LIN {X 0,Y 148.695,Z 336.424,A -85,B 0,C 180,E1 -24524.199,E2 -24524.199} C_VEL
LIN {X 0,Y 149.937,Z 338.136,A -85,B 0,C 180,E1 -24524.799,E2 -24524.799} C_VEL
LIN {X 0,Y 154.81,Z 345.559,A -85,B 0,C 180,E1 -24527.052,E2 -24527.052} C_VEL
LIN {X 0,Y 158.039,Z 351.12,A -85,B 0,C 180,E1 -24528.465,E2 -24528.465} C_VEL
LIN {X 0,Y 163.343,Z 362.974,A -85,B 0,C 180,E1 -24530.756,E2 -24530.756} C_VEL
LIN {X 0,Y 166.745,Z 372.421,A -85,B 0,C 180,E1 -24532.212,E2 -24532.212} C_VEL
LIN {X 0,Y 166.413,Z 382.188,A -85,B 0,C 180,E1 -24532.644,E2 -24532.644} C_VEL
LIN {X 0,Y 165.211,Z 401.171,A -85,B 0,C 180,E1 -24533.449,E2 -24533.449} C_VEL
LIN {X 0,Y 163.851,Z 412.228,A -85,B 0,C 180,E1 -24534.244,E2 -24534.244} C_VEL
LIN {X 0,Y 161.723,Z 423.778,A -85,B 0,C 180,E1 -24535.603,E2 -24535.603} C_VEL
LIN {X 0,Y 159.816,Z 431.992,A -85,B 0,C 180,E1 -24536.921,E2 -24536.921} C_VEL
LIN {X 0,Y 157.688,Z 439.473,A -85,B 0,C 180,E1 -24538.421,E2 -24538.421} C_VEL
LIN {X 0,Y 155.05,Z 447.512,A -85,B 0,C 180,E1 -24540.467,E2 -24540.467} C_VEL
LIN {X 0,Y 152.63,Z 454.152,A -85,B 0,C 180,E1 -24542.584,E2 -24542.584} C_VEL
LIN {X 0,Y 150.051,Z 460.455,A -85,B 0,C 180,E1 -24545.069,E2 -24545.069} C_VEL
LIN {X 0,Y 147.775,Z 465.69,A -85,B 0,C 180,E1 -24547.638,E2 -24547.638} C_VEL
LIN {X 0,Y 145.868,Z 470.055,A -85,B 0,C 180,E1 -24550.29,E2 -24550.29} C_VEL
LIN {X 0,Y 143.545,Z 475.202,A -85,B 0,C 180,E1 -24554.379,E2 -24554.379} C_VEL
LIN {X 0,Y 141.917,Z 478.977,A -85,B 0,C 180,E1 -24558.575,E2 -24558.575} C_VEL
LIN {X 0,Y 141.219,Z 480.707,A -85,B 0,C 180,E1 -24561.414,E2 -24561.414} C_VEL
LIN {X 0,Y 140.732,Z 481.944,A -85,B 0,C 180,E1 -24564.268,E2 -24564.268} C_VEL
LIN {X 0,Y 140.537,Z 482.711,A -85,B 0,C 180,E1 -24567.134,E2 -24567.134} C_VEL
LIN {X 0,Y 140.501,Z 483,A -85,B 0,C 180,E1 -24570,E2 -24570} C_VEL
LIN {X 0,Y 140.537,Z 482.7,A -85,B 0,C 180,E1 -24572.866,E2 -24572.866} C_VEL
LIN {X 0,Y 140.727,Z 481.911,A -85,B 0,C 180,E1 -24575.732,E2 -24575.732} C_VEL
LIN {X 0,Y 141.165,Z 480.651,A -85,B 0,C 180,E1 -24578.589,E2 -24578.589} C_VEL
LIN {X 0,Y 142.391,Z 477.747,A -85,B 0,C 180,E1 -24582.832,E2 -24582.832} C_VEL
LIN {X 0,Y 143.538,Z 475.097,A -85,B 0,C 180,E1 -24585.622,E2 -24585.622} C_VEL
LIN {X 0,Y 145.852,Z 469.92,A -85,B 0,C 180,E1 -24589.712,E2 -24589.712} C_VEL
LIN {X 0,Y 147.47,Z 466.222,A -85,B 0,C 180,E1 -24591.972,E2 -24591.972} C_VEL
LIN {X 0,Y 148.291,Z 462.951,A -85,B 0,C 180,E1 -24593.828,E2 -24593.828} C_VEL
LIN {X 0,Y 148.181,Z 457.047,A -85,B 0,C 180,E1 -24596.903,E2 -24596.903} C_VEL
LIN {X 0,Y 148.279,Z 450.489,A -85,B 0,C 180,E1 -24599.774,E2 -24599.774} C_VEL
LIN {X 0,Y 149.393,Z 445.99,A -85,B 0,C 180,E1 -24601.248,E2 -24601.248} C_VEL
LIN {X 0,Y 152.515,Z 436.512,A -85,B 0,C 180,E1 -24603.57,E2 -24603.57} C_VEL
LIN {X 0,Y 154.97,Z 427.195,A -85,B 0,C 180,E1 -24605.283,E2 -24605.283} C_VEL
LIN {X 0,Y 157.011,Z 417.741,A -85,B 0,C 180,E1 -24606.577,E2 -24606.577} C_VEL
LIN {X 0,Y 158.536,Z 408.45,A -85,B 0,C 180,E1 -24607.495,E2 -24607.495} C_VEL
LIN {X 0,Y 159.576,Z 399.713,A -85,B 0,C 180,E1 -24608.066,E2 -24608.066} C_VEL
LIN {X 0,Y 161.057,Z 374.2,A -85,B 0,C 180,E1 -24609.16,E2 -24609.16} C_VEL
LIN {X 0,Y 156.299,Z 361.781,A -85,B 0,C 180,E1 -24611.334,E2 -24611.334} C_VEL
LIN {X 0,Y 152.216,Z 352.913,A -85,B 0,C 180,E1 -24613.26,E2 -24613.26} C_VEL
LIN {X 0,Y 145.462,Z 342.285,A -85,B 0,C 180,E1 -24616.558,E2 -24616.558} C_VEL
LIN {X 0,Y 142.86,Z 338.543,A -85,B 0,C 180,E1 -24617.945,E2 -24617.945} C_VEL
LIN {X 0,Y 140.098,Z 334.863,A -85,B 0,C 180,E1 -24619.495,E2 -24619.495} C_VEL
LIN {X 0,Y 139.28,Z 333.439,A -85,B 0,C 180,E1 -24620.002,E2 -24620.002} C_VEL
LIN {X 0,Y 137.047,Z 331.169,A -85,B 0,C 180,E1 -24621.313,E2 -24621.313} C_VEL
LIN {X 0,Y 136.131,Z 328.935,A -85,B 0,C 180,E1 -24622.189,E2 -24622.189} C_VEL
LIN {X 0,Y 136.019,Z 328.352,A -85,B 0,C 180,E1 -24623.083,E2 -24623.083} C_VEL
LIN {X 0,Y 136.079,Z 328.326,A -85,B 0,C 180,E1 -24625.723,E2 -24625.723} C_VEL
LIN {X 0,Y 136.114,Z 328.328,A -85,B 0,C 180,E1 -24632.31,E2 -24632.31} C_VEL
LIN {X 0,Y 136.18,Z 328.306,A -85,B 0,C 180,E1 -24638.823,E2 -24638.823} C_VEL
LIN {X 0,Y 136.218,Z 328.297,A -85,B 0,C 180,E1 -24645.051,E2 -24645.051} C_VEL
LIN {X 0,Y 136.422,Z 328.278,A -85,B 0,C 180,E1 -24648.179,E2 -24648.179} C_VEL
LIN {X 0,Y 136.541,Z 328.288,A -85,B 0,C 180,E1 -24651.117,E2 -24651.117} C_VEL
LIN {X 0,Y 137.105,Z 328.22,A -85,B 0,C 180,E1 -24660,E2 -24660} C_VEL
LIN {X 0,Y 136.529,Z 328.289,A -85,B 0,C 180,E1 -24668.884,E2 -24668.884} C_VEL
LIN {X 0,Y 136.41,Z 328.279,A -85,B 0,C 180,E1 -24671.893,E2 -24671.893} C_VEL
LIN {X 0,Y 136.162,Z 328.337,A -85,B 0,C 180,E1 -24678.041,E2 -24678.041} C_VEL
LIN {X 0,Y 136.143,Z 328.308,A -85,B 0,C 180,E1 -24681.693,E2 -24681.693} C_VEL
LIN {X 0,Y 136.085,Z 328.324,A -85,B 0,C 180,E1 -24688.606,E2 -24688.606} C_VEL
LIN {X 0,Y 136.066,Z 328.321,A -85,B 0,C 180,E1 -24694.623,E2 -24694.623} C_VEL
LIN {X 0,Y 136.059,Z 328.636,A -85,B 0,C 180,E1 -24697.544,E2 -24697.544} C_VEL
LIN {X 0,Y 136.414,Z 329.867,A -85,B 0,C 180,E1 -24698.264,E2 -24698.264} C_VEL
LIN {X 0,Y 138.033,Z 332.419,A -85,B 0,C 180,E1 -24699.341,E2 -24699.341} C_VEL
LIN {X 0,Y 139.651,Z 333.976,A -85,B 0,C 180,E1 -24700.266,E2 -24700.266} C_VEL
LIN {X 0,Y 141.692,Z 337.197,A -85,B 0,C 180,E1 -24701.474,E2 -24701.474} C_VEL
LIN {X 0,Y 142.993,Z 338.765,A -85,B 0,C 180,E1 -24702.175,E2 -24702.175} C_VEL
LIN {X 0,Y 148.809,Z 347.525,A -85,B 0,C 180,E1 -24705.181,E2 -24705.181} C_VEL
LIN {X 0,Y 153.169,Z 354.766,A -85,B 0,C 180,E1 -24707.235,E2 -24707.235} C_VEL
LIN {X 0,Y 157.306,Z 364.284,A -85,B 0,C 180,E1 -24709.18,E2 -24709.18} C_VEL
LIN {X 0,Y 161.073,Z 374.306,A -85,B 0,C 180,E1 -24710.895,E2 -24710.895} C_VEL
LIN {X 0,Y 159.461,Z 400.566,A -85,B 0,C 180,E1 -24712.012,E2 -24712.012} C_VEL
LIN {X 0,Y 158.152,Z 411.086,A -85,B 0,C 180,E1 -24712.761,E2 -24712.761} C_VEL
LIN {X 0,Y 155.974,Z 423.044,A -85,B 0,C 180,E1 -24714.144,E2 -24714.144} C_VEL
LIN {X 0,Y 153.613,Z 432.702,A -85,B 0,C 180,E1 -24715.745,E2 -24715.745} C_VEL
LIN {X 0,Y 151.353,Z 440.221,A -85,B 0,C 180,E1 -24717.331,E2 -24717.331} C_VEL
LIN {X 0,Y 148.95,Z 447.117,A -85,B 0,C 180,E1 -24719.129,E2 -24719.129} C_VEL
LIN {X 0,Y 146.422,Z 453.821,A -85,B 0,C 180,E1 -24721.317,E2 -24721.317} C_VEL
LIN {X 0,Y 143.695,Z 460.173,A -85,B 0,C 180,E1 -24723.885,E2 -24723.885} C_VEL
LIN {X 0,Y 141.259,Z 465.454,A -85,B 0,C 180,E1 -24726.546,E2 -24726.546} C_VEL
LIN {X 0,Y 139.225,Z 469.863,A -85,B 0,C 180,E1 -24729.308,E2 -24729.308} C_VEL
LIN {X 0,Y 136.733,Z 475.052,A -85,B 0,C 180,E1 -24733.579,E2 -24733.579} C_VEL
LIN {X 0,Y 135.505,Z 477.712,A -85,B 0,C 180,E1 -24736.503,E2 -24736.503} C_VEL
LIN {X 0,Y 134.143,Z 480.627,A -85,B 0,C 180,E1 -24740.957,E2 -24740.957} C_VEL
LIN {X 0,Y 133.662,Z 481.896,A -85,B 0,C 180,E1 -24743.964,E2 -24743.964} C_VEL
LIN {X 0,Y 133.466,Z 482.695,A -85,B 0,C 180,E1 -24746.982,E2 -24746.982} C_VEL
LIN {X 0,Y 133.419,Z 482.999,A -85,B 0,C 180,E1 -24750,E2 -24750} C_VEL
LIN {X 0,Y 133.466,Z 482.716,A -85,B 0,C 180,E1 -24753.018,E2 -24753.018} C_VEL
LIN {X 0,Y 133.662,Z 481.959,A -85,B 0,C 180,E1 -24756.036,E2 -24756.036} C_VEL
LIN {X 0,Y 134.142,Z 480.732,A -85,B 0,C 180,E1 -24759.043,E2 -24759.043} C_VEL
LIN {X 0,Y 135.48,Z 477.861,A -85,B 0,C 180,E1 -24763.499,E2 -24763.499} C_VEL
LIN {X 0,Y 136.68,Z 475.247,A -85,B 0,C 180,E1 -24766.427,E2 -24766.427} C_VEL
LIN {X 0,Y 139.185,Z 470.112,A -85,B 0,C 180,E1 -24770.698,E2 -24770.698} C_VEL
LIN {X 0,Y 141.795,Z 464.588,A -85,B 0,C 180,E1 -24774.136,E2 -24774.136} C_VEL
LIN {X 0,Y 144.923,Z 457.644,A -85,B 0,C 180,E1 -24777.432,E2 -24777.432} C_VEL
LIN {X 0,Y 148.155,Z 449.673,A -85,B 0,C 180,E1 -24780.265,E2 -24780.265} C_VEL
LIN {X 0,Y 150.871,Z 442.075,A -85,B 0,C 180,E1 -24782.391,E2 -24782.391} C_VEL
LIN {X 0,Y 153.042,Z 435.345,A -85,B 0,C 180,E1 -24783.903,E2 -24783.903} C_VEL
LIN {X 0,Y 155.42,Z 426.284,A -85,B 0,C 180,E1 -24785.516,E2 -24785.516} C_VEL
LIN {X 0,Y 157.213,Z 417.303,A -85,B 0,C 180,E1 -24786.753,E2 -24786.753} C_VEL
LIN {X 0,Y 158.785,Z 407.979,A -85,B 0,C 180,E1 -24787.641,E2 -24787.641} C_VEL
LIN {X 0,Y 159.771,Z 398.211,A -85,B 0,C 180,E1 -24788.286,E2 -24788.286} C_VEL
LIN {X 0,Y 161.177,Z 374.379,A -85,B 0,C 180,E1 -24789.275,E2 -24789.275} C_VEL
LIN {X 0,Y 156.324,Z 361.554,A -85,B 0,C 180,E1 -24791.51,E2 -24791.51} C_VEL
LIN {X 0,Y 152.125,Z 352.746,A -85,B 0,C 180,E1 -24793.483,E2 -24793.483} C_VEL
LIN {X 0,Y 145.533,Z 342.329,A -85,B 0,C 180,E1 -24796.725,E2 -24796.725} C_VEL
LIN {X 0,Y 142.997,Z 338.745,A -85,B 0,C 180,E1 -24798.077,E2 -24798.077} C_VEL
LIN {X 0,Y 140.121,Z 334.906,A -85,B 0,C 180,E1 -24799.7,E2 -24799.7} C_VEL
LIN {X 0,Y 139.31,Z 333.464,A -85,B 0,C 180,E1 -24800.208,E2 -24800.208} C_VEL
LIN {X 0,Y 137.107,Z 331.257,A -85,B 0,C 180,E1 -24801.507,E2 -24801.507} C_VEL
LIN {X 0,Y 136.142,Z 328.931,A -85,B 0,C 180,E1 -24802.425,E2 -24802.425} C_VEL
LIN {X 0,Y 136.037,Z 328.331,A -85,B 0,C 180,E1 -24803.55,E2 -24803.55} C_VEL
LIN {X 0,Y 136.051,Z 328.33,A -85,B 0,C 180,E1 -24808.897,E2 -24808.897} C_VEL
LIN {X 0,Y 136.115,Z 328.326,A -85,B 0,C 180,E1 -24812.309,E2 -24812.309} C_VEL
LIN {X 0,Y 136.181,Z 328.305,A -85,B 0,C 180,E1 -24818.822,E2 -24818.822} C_VEL
LIN {X 0,Y 136.218,Z 328.298,A -85,B 0,C 180,E1 -24825.05,E2 -24825.05} C_VEL
LIN {X 0,Y 136.423,Z 328.277,A -85,B 0,C 180,E1 -24828.178,E2 -24828.178} C_VEL
LIN {X 0,Y 136.541,Z 328.288,A -85,B 0,C 180,E1 -24831.117,E2 -24831.117} C_VEL
LIN {X 0,Y 137.105,Z 328.22,A -85,B 0,C 180,E1 -24840,E2 -24840} C_VEL
LIN {X 0,Y 136.529,Z 328.289,A -85,B 0,C 180,E1 -24848.883,E2 -24848.883} C_VEL
LIN {X 0,Y 136.41,Z 328.278,A -85,B 0,C 180,E1 -24851.893,E2 -24851.893} C_VEL
LIN {X 0,Y 136.161,Z 328.337,A -85,B 0,C 180,E1 -24858.04,E2 -24858.04} C_VEL
LIN {X 0,Y 136.143,Z 328.308,A -85,B 0,C 180,E1 -24861.693,E2 -24861.693} C_VEL
LIN {X 0,Y 136.084,Z 328.323,A -85,B 0,C 180,E1 -24868.605,E2 -24868.605} C_VEL
LIN {X 0,Y 136.043,Z 328.32,A -85,B 0,C 180,E1 -24874.629,E2 -24874.629} C_VEL
LIN {X 0,Y 136.057,Z 328.64,A -85,B 0,C 180,E1 -24877.31,E2 -24877.31} C_VEL
LIN {X 0,Y 136.449,Z 329.96,A -85,B 0,C 180,E1 -24878.058,E2 -24878.058} C_VEL
LIN {X 0,Y 138.064,Z 332.476,A -85,B 0,C 180,E1 -24879.133,E2 -24879.133} C_VEL
LIN {X 0,Y 139.681,Z 333.957,A -85,B 0,C 180,E1 -24880.058,E2 -24880.058} C_VEL
LIN {X 0,Y 141.743,Z 337.249,A -85,B 0,C 180,E1 -24881.288,E2 -24881.288} C_VEL
LIN {X 0,Y 143.034,Z 338.862,A -85,B 0,C 180,E1 -24881.993,E2 -24881.993} C_VEL
LIN {X 0,Y 148.483,Z 346.884,A -85,B 0,C 180,E1 -24884.822,E2 -24884.822} C_VEL
LIN {X 0,Y 153.376,Z 355.105,A -85,B 0,C 180,E1 -24887.151,E2 -24887.151} C_VEL
LIN {X 0,Y 158.553,Z 367.079,A -85,B 0,C 180,E1 -24889.566,E2 -24889.566} C_VEL
LIN {X 0,Y 161.175,Z 374.479,A -85,B 0,C 180,E1 -24890.775,E2 -24890.775} C_VEL
LIN {X 0,Y 159.576,Z 401.187,A -85,B 0,C 180,E1 -24891.934,E2 -24891.934} C_VEL
LIN {X 0,Y 158.064,Z 412.877,A -85,B 0,C 180,E1 -24892.806,E2 -24892.806} C_VEL
LIN {X 0,Y 155.92,Z 423.784,A -85,B 0,C 180,E1 -24894.13,E2 -24894.13} C_VEL
LIN {X 0,Y 153.706,Z 432.765,A -85,B 0,C 180,E1 -24895.628,E2 -24895.628} C_VEL
LIN {X 0,Y 151.277,Z 440.706,A -85,B 0,C 180,E1 -24897.312,E2 -24897.312} C_VEL
LIN {X 0,Y 148.545,Z 448.536,A -85,B 0,C 180,E1 -24899.43,E2 -24899.43} C_VEL
LIN {X 0,Y 145.646,Z 455.858,A -85,B 0,C 180,E1 -24901.936,E2 -24901.936} C_VEL
LIN {X 0,Y 142.4,Z 463.284,A -85,B 0,C 180,E1 -24905.197,E2 -24905.197} C_VEL
LIN {X 0,Y 139.71,Z 469.1,A -85,B 0,C 180,E1 -24908.611,E2 -24908.611} C_VEL
LIN {X 0,Y 137.458,Z 473.686,A -85,B 0,C 180,E1 -24912.136,E2 -24912.136} C_VEL
LIN {X 0,Y 136.064,Z 476.666,A -85,B 0,C 180,E1 -24915.034,E2 -24915.034} C_VEL
LIN {X 0,Y 134.962,Z 478.978,A -85,B 0,C 180,E1 -24917.978,E2 -24917.978} C_VEL
LIN {X 0,Y 134.184,Z 480.708,A -85,B 0,C 180,E1 -24920.96,E2 -24920.96} C_VEL
LIN {X 0,Y 133.667,Z 481.945,A -85,B 0,C 180,E1 -24923.964,E2 -24923.964} C_VEL
LIN {X 0,Y 133.464,Z 482.711,A -85,B 0,C 180,E1 -24926.982,E2 -24926.982} C_VEL
LIN {X 0,Y 133.418,Z 483,A -85,B 0,C 180,E1 -24930,E2 -24930} C_VEL
LIN {X 0,Y 133.464,Z 482.7,A -85,B 0,C 180,E1 -24933.018,E2 -24933.018} C_VEL
LIN {X 0,Y 133.661,Z 481.911,A -85,B 0,C 180,E1 -24936.036,E2 -24936.036} C_VEL
LIN {X 0,Y 134.141,Z 480.651,A -85,B 0,C 180,E1 -24939.043,E2 -24939.043} C_VEL
LIN {X 0,Y 135.482,Z 477.746,A -85,B 0,C 180,E1 -24943.499,E2 -24943.499} C_VEL
LIN {X 0,Y 136.7,Z 475.096,A -85,B 0,C 180,E1 -24946.425,E2 -24946.425} C_VEL
LIN {X 0,Y 139.176,Z 469.919,A -85,B 0,C 180,E1 -24950.7,E2 -24950.7} C_VEL
LIN {X 0,Y 142.4,Z 463.086,A -85,B 0,C 180,E1 -24954.803,E2 -24954.803} C_VEL
LIN {X 0,Y 145.648,Z 455.62,A -85,B 0,C 180,E1 -24958.064,E2 -24958.064} C_VEL
LIN {X 0,Y 148.533,Z 448.254,A -85,B 0,C 180,E1 -24960.573,E2 -24960.573} C_VEL
LIN {X 0,Y 149.393,Z 445.99,A -85,B 0,C 180,E1 -24961.248,E2 -24961.248} C_VEL
LIN {X 0,Y 150.48,Z 441.43,A -85,B 0,C 180,E1 -24962.633,E2 -24962.633} C_VEL
LIN {X 0,Y 150.534,Z 433.661,A -85,B 0,C 180,E1 -24964.998,E2 -24964.998} C_VEL
LIN {X 0,Y 150.331,Z 425.341,A -85,B 0,C 180,E1 -24967.057,E2 -24967.057} C_VEL
LIN {X 0,Y 150.947,Z 419.921,A -85,B 0,C 180,E1 -24967.922,E2 -24967.922} C_VEL
LIN {X 0,Y 152.843,Z 409.396,A -85,B 0,C 180,E1 -24969.029,E2 -24969.029} C_VEL
LIN {X 0,Y 154.058,Z 399.697,A -85,B 0,C 180,E1 -24969.691,E2 -24969.691} C_VEL
LIN {X 0,Y 155.493,Z 376.136,A -85,B 0,C 180,E1 -24970.733,E2 -24970.733} C_VEL
LIN {X 0,Y 151.514,Z 365.491,A -85,B 0,C 180,E1 -24972.71,E2 -24972.71} C_VEL
LIN {X 0,Y 147.907,Z 357.529,A -85,B 0,C 180,E1 -24974.542,E2 -24974.542} C_VEL
LIN {X 0,Y 141.823,Z 347.659,A -85,B 0,C 180,E1 -24977.734,E2 -24977.734} C_VEL
LIN {X 0,Y 138.092,Z 342.464,A -85,B 0,C 180,E1 -24979.874,E2 -24979.874} C_VEL
LIN {X 0,Y 135.728,Z 338.996,A -85,B 0,C 180,E1 -24981.359,E2 -24981.359} C_VEL
LIN {X 0,Y 133.34,Z 335.935,A -85,B 0,C 180,E1 -24982.927,E2 -24982.927} C_VEL
LIN {X 0,Y 132.436,Z 334.429,A -85,B 0,C 180,E1 -24983.581,E2 -24983.581} C_VEL
LIN {X 0,Y 130.24,Z 332.395,A -85,B 0,C 180,E1 -24985.103,E2 -24985.103} C_VEL
LIN {X 0,Y 129.116,Z 329.851,A -85,B 0,C 180,E1 -24986.308,E2 -24986.308} C_VEL
LIN {X 0,Y 128.997,Z 329.255,A -85,B 0,C 180,E1 -24987.452,E2 -24987.452} C_VEL
LIN {X 0,Y 129.014,Z 329.201,A -85,B 0,C 180,E1 -24990.642,E2 -24990.642} C_VEL
LIN {X 0,Y 128.995,Z 329.229,A -85,B 0,C 180,E1 -24994.16,E2 -24994.16} C_VEL
LIN {X 0,Y 129.065,Z 329.188,A -85,B 0,C 180,E1 -24997.771,E2 -24997.771} C_VEL
LIN {X 0,Y 129.141,Z 329.184,A -85,B 0,C 180,E1 -25004.211,E2 -25004.211} C_VEL
LIN {X 0,Y 129.34,Z 329.156,A -85,B 0,C 180,E1 -25007.974,E2 -25007.974} C_VEL
LIN {X 0,Y 129.465,Z 329.17,A -85,B 0,C 180,E1 -25010.628,E2 -25010.628} C_VEL
LIN {X 0,Y 130.06,Z 329.098,A -85,B 0,C 180,E1 -25020,E2 -25020} C_VEL
LIN {X 0,Y 129.456,Z 329.171,A -85,B 0,C 180,E1 -25029.374,E2 -25029.374} C_VEL
LIN {X 0,Y 129.294,Z 329.158,A -85,B 0,C 180,E1 -25032.558,E2 -25032.558} C_VEL
LIN {X 0,Y 129.079,Z 329.211,A -85,B 0,C 180,E1 -25039.068,E2 -25039.068} C_VEL
LIN {X 0,Y 129.039,Z 329.192,A -85,B 0,C 180,E1 -25042.411,E2 -25042.411} C_VEL
LIN {X 0,Y 128.995,Z 329.228,A -85,B 0,C 180,E1 -25045.84,E2 -25045.84} C_VEL
LIN {X 0,Y 129.001,Z 329.207,A -85,B 0,C 180,E1 -25051.169,E2 -25051.169} C_VEL
LIN {X 0,Y 129.048,Z 329.596,A -85,B 0,C 180,E1 -25053.474,E2 -25053.474} C_VEL
LIN {X 0,Y 129.49,Z 330.922,A -85,B 0,C 180,E1 -25054.3,E2 -25054.3} C_VEL
LIN {X 0,Y 131.021,Z 333.346,A -85,B 0,C 180,E1 -25055.516,E2 -25055.516} C_VEL
LIN {X 0,Y 132.865,Z 334.901,A -85,B 0,C 180,E1 -25056.755,E2 -25056.755} C_VEL
LIN {X 0,Y 134.824,Z 338.072,A -85,B 0,C 180,E1 -25058.126,E2 -25058.126} C_VEL
LIN {X 0,Y 136.468,Z 339.947,A -85,B 0,C 180,E1 -25059.151,E2 -25059.151} C_VEL
LIN {X 0,Y 138.92,Z 343.431,A -85,B 0,C 180,E1 -25060.649,E2 -25060.649} C_VEL
LIN {X 0,Y 144.623,Z 352.07,A -85,B 0,C 180,E1 -25063.827,E2 -25063.827} C_VEL
LIN {X 0,Y 148.928,Z 359.491,A -85,B 0,C 180,E1 -25066.017,E2 -25066.017} C_VEL
LIN {X 0,Y 153.362,Z 370.157,A -85,B 0,C 180,E1 -25068.256,E2 -25068.256} C_VEL
LIN {X 0,Y 155.505,Z 376.196,A -85,B 0,C 180,E1 -25069.319,E2 -25069.319} C_VEL
LIN {X 0,Y 153.894,Z 401.036,A -85,B 0,C 180,E1 -25070.413,E2 -25070.413} C_VEL
LIN {X 0,Y 152.457,Z 411.896,A -85,B 0,C 180,E1 -25071.218,E2 -25071.218} C_VEL
LIN {X 0,Y 150.279,Z 423.05,A -85,B 0,C 180,E1 -25072.559,E2 -25072.559} C_VEL
LIN {X 0,Y 147.966,Z 432.158,A -85,B 0,C 180,E1 -25074.089,E2 -25074.089} C_VEL
LIN {X 0,Y 145.441,Z 440.225,A -85,B 0,C 180,E1 -25075.825,E2 -25075.825} C_VEL
LIN {X 0,Y 142.892,Z 447.12,A -85,B 0,C 180,E1 -25077.665,E2 -25077.665} C_VEL
LIN {X 0,Y 140.247,Z 453.824,A -85,B 0,C 180,E1 -25079.927,E2 -25079.927} C_VEL
LIN {X 0,Y 137.352,Z 460.176,A -85,B 0,C 180,E1 -25082.581,E2 -25082.581} C_VEL
LIN {X 0,Y 134.779,Z 465.456,A -85,B 0,C 180,E1 -25085.345,E2 -25085.345} C_VEL
LIN {X 0,Y 132.592,Z 469.865,A -85,B 0,C 180,E1 -25088.221,E2 -25088.221} C_VEL
LIN {X 0,Y 129.931,Z 475.053,A -85,B 0,C 180,E1 -25092.693,E2 -25092.693} C_VEL
LIN {X 0,Y 128.595,Z 477.713,A -85,B 0,C 180,E1 -25095.763,E2 -25095.763} C_VEL
LIN {X 0,Y 127.143,Z 480.627,A -85,B 0,C 180,E1 -25100.455,E2 -25100.455} C_VEL
LIN {X 0,Y 126.595,Z 481.897,A -85,B 0,C 180,E1 -25103.625,E2 -25103.625} C_VEL
LIN {X 0,Y 126.382,Z 482.695,A -85,B 0,C 180,E1 -25106.812,E2 -25106.812} C_VEL
LIN {X 0,Y 126.322,Z 482.999,A -85,B 0,C 180,E1 -25110,E2 -25110} C_VEL
LIN {X 0,Y 126.382,Z 482.716,A -85,B 0,C 180,E1 -25113.188,E2 -25113.188} C_VEL
LIN {X 0,Y 126.595,Z 481.959,A -85,B 0,C 180,E1 -25116.375,E2 -25116.375} C_VEL
LIN {X 0,Y 127.142,Z 480.731,A -85,B 0,C 180,E1 -25119.545,E2 -25119.545} C_VEL
LIN {X 0,Y 128.57,Z 477.86,A -85,B 0,C 180,E1 -25124.24,E2 -25124.24} C_VEL
LIN {X 0,Y 129.883,Z 475.246,A -85,B 0,C 180,E1 -25127.314,E2 -25127.314} C_VEL
LIN {X 0,Y 132.555,Z 470.11,A -85,B 0,C 180,E1 -25131.785,E2 -25131.785} C_VEL
LIN {X 0,Y 135.33,Z 464.586,A -85,B 0,C 180,E1 -25135.368,E2 -25135.368} C_VEL
LIN {X 0,Y 138.659,Z 457.641,A -85,B 0,C 180,E1 -25138.783,E2 -25138.783} C_VEL
LIN {X 0,Y 142.064,Z 449.67,A -85,B 0,C 180,E1 -25141.709,E2 -25141.709} C_VEL
LIN {X 0,Y 144.94,Z 442.071,A -85,B 0,C 180,E1 -25143.891,E2 -25143.891} C_VEL
LIN {X 0,Y 147.528,Z 434.049,A -85,B 0,C 180,E1 -25145.716,E2 -25145.716} C_VEL
LIN {X 0,Y 149.854,Z 425.655,A -85,B 0,C 180,E1 -25147.19,E2 -25147.19} C_VEL
LIN {X 0,Y 151.7,Z 416.639,A -85,B 0,C 180,E1 -25148.439,E2 -25148.439} C_VEL
LIN {X 0,Y 153.358,Z 406.897,A -85,B 0,C 180,E1 -25149.359,E2 -25149.359} C_VEL
LIN {X 0,Y 154.572,Z 394.44,A -85,B 0,C 180,E1 -25150.102,E2 -25150.102} C_VEL
LIN {X 0,Y 155.669,Z 376.382,A -85,B 0,C 180,E1 -25150.832,E2 -25150.832} C_VEL
LIN {X 0,Y 151.079,Z 364.134,A -85,B 0,C 180,E1 -25153.129,E2 -25153.129} C_VEL
LIN {X 0,Y 147.817,Z 357.328,A -85,B 0,C 180,E1 -25154.779,E2 -25154.779} C_VEL
LIN {X 0,Y 141.871,Z 347.69,A -85,B 0,C 180,E1 -25157.92,E2 -25157.92} C_VEL
LIN {X 0,Y 138.318,Z 342.743,A -85,B 0,C 180,E1 -25159.965,E2 -25159.965} C_VEL
LIN {X 0,Y 135.902,Z 339.167,A -85,B 0,C 180,E1 -25161.488,E2 -25161.488} C_VEL
LIN {X 0,Y 133.584,Z 336.285,A -85,B 0,C 180,E1 -25163.005,E2 -25163.005} C_VEL
LIN {X 0,Y 132.702,Z 334.585,A -85,B 0,C 180,E1 -25163.665,E2 -25163.665} C_VEL
LIN {X 0,Y 130.37,Z 332.591,A -85,B 0,C 180,E1 -25165.27,E2 -25165.27} C_VEL
LIN {X 0,Y 129.117,Z 329.902,A -85,B 0,C 180,E1 -25166.55,E2 -25166.55} C_VEL
LIN {X 0,Y 128.989,Z 329.282,A -85,B 0,C 180,E1 -25167.449,E2 -25167.449} C_VEL
LIN {X 0,Y 129.015,Z 329.2,A -85,B 0,C 180,E1 -25170.641,E2 -25170.641} C_VEL
LIN {X 0,Y 128.995,Z 329.23,A -85,B 0,C 180,E1 -25174.16,E2 -25174.16} C_VEL
LIN {X 0,Y 129.066,Z 329.188,A -85,B 0,C 180,E1 -25177.77,E2 -25177.77} C_VEL
LIN {X 0,Y 129.141,Z 329.185,A -85,B 0,C 180,E1 -25184.21,E2 -25184.21} C_VEL
LIN {X 0,Y 129.34,Z 329.156,A -85,B 0,C 180,E1 -25187.973,E2 -25187.973} C_VEL
LIN {X 0,Y 129.465,Z 329.17,A -85,B 0,C 180,E1 -25190.627,E2 -25190.627} C_VEL
LIN {X 0,Y 130.06,Z 329.098,A -85,B 0,C 180,E1 -25200,E2 -25200} C_VEL
LIN {X 0,Y 129.456,Z 329.171,A -85,B 0,C 180,E1 -25209.373,E2 -25209.373} C_VEL
LIN {X 0,Y 129.294,Z 329.158,A -85,B 0,C 180,E1 -25212.558,E2 -25212.558} C_VEL
LIN {X 0,Y 129.078,Z 329.21,A -85,B 0,C 180,E1 -25219.067,E2 -25219.067} C_VEL
LIN {X 0,Y 129.039,Z 329.192,A -85,B 0,C 180,E1 -25222.411,E2 -25222.411} C_VEL
LIN {X 0,Y 128.995,Z 329.229,A -85,B 0,C 180,E1 -25225.84,E2 -25225.84} C_VEL
LIN {X 0,Y 128.999,Z 329.208,A -85,B 0,C 180,E1 -25231.169,E2 -25231.169} C_VEL
LIN {X 0,Y 129.054,Z 329.632,A -85,B 0,C 180,E1 -25233.231,E2 -25233.231} C_VEL
LIN {X 0,Y 129.501,Z 331.019,A -85,B 0,C 180,E1 -25234.047,E2 -25234.047} C_VEL
LIN {X 0,Y 131.127,Z 333.468,A -85,B 0,C 180,E1 -25235.331,E2 -25235.331} C_VEL
LIN {X 0,Y 132.878,Z 334.934,A -85,B 0,C 180,E1 -25236.514,E2 -25236.514} C_VEL
LIN {X 0,Y 134.946,Z 338.233,A -85,B 0,C 180,E1 -25237.966,E2 -25237.966} C_VEL
LIN {X 0,Y 136.51,Z 339.967,A -85,B 0,C 180,E1 -25238.942,E2 -25238.942} C_VEL
LIN {X 0,Y 139.13,Z 343.65,A -85,B 0,C 180,E1 -25240.547,E2 -25240.547} C_VEL
LIN {X 0,Y 145.208,Z 353.043,A -85,B 0,C 180,E1 -25243.938,E2 -25243.938} C_VEL
LIN {X 0,Y 149.028,Z 359.63,A -85,B 0,C 180,E1 -25245.878,E2 -25245.878} C_VEL
LIN {X 0,Y 153.69,Z 370.747,A -85,B 0,C 180,E1 -25248.227,E2 -25248.227} C_VEL
LIN {X 0,Y 155.657,Z 376.357,A -85,B 0,C 180,E1 -25249.207,E2 -25249.207} C_VEL
LIN {X 0,Y 154.056,Z 401.203,A -85,B 0,C 180,E1 -25250.308,E2 -25250.308} C_VEL
LIN {X 0,Y 152.547,Z 412.321,A -85,B 0,C 180,E1 -25251.134,E2 -25251.134} C_VEL
LIN {X 0,Y 150.239,Z 423.79,A -85,B 0,C 180,E1 -25252.547,E2 -25252.547} C_VEL
LIN {X 0,Y 147.893,Z 432.773,A -85,B 0,C 180,E1 -25254.074,E2 -25254.074} C_VEL
LIN {X 0,Y 145.362,Z 440.71,A -85,B 0,C 180,E1 -25255.803,E2 -25255.803} C_VEL
LIN {X 0,Y 142.474,Z 448.539,A -85,B 0,C 180,E1 -25257.977,E2 -25257.977} C_VEL
LIN {X 0,Y 139.43,Z 455.861,A -85,B 0,C 180,E1 -25260.565,E2 -25260.565} C_VEL
LIN {X 0,Y 135.987,Z 463.286,A -85,B 0,C 180,E1 -25263.942,E2 -25263.942} C_VEL
LIN {X 0,Y 133.117,Z 469.102,A -85,B 0,C 180,E1 -25267.495,E2 -25267.495} C_VEL
LIN {X 0,Y 130.711,Z 473.687,A -85,B 0,C 180,E1 -25271.18,E2 -25271.18} C_VEL
LIN {X 0,Y 129.197,Z 476.667,A -85,B 0,C 180,E1 -25274.218,E2 -25274.218} C_VEL
LIN {X 0,Y 128.012,Z 478.979,A -85,B 0,C 180,E1 -25277.314,E2 -25277.314} C_VEL
LIN {X 0,Y 127.173,Z 480.709,A -85,B 0,C 180,E1 -25280.457,E2 -25280.457} C_VEL
LIN {X 0,Y 126.599,Z 481.945,A -85,B 0,C 180,E1 -25283.626,E2 -25283.626} C_VEL
LIN {X 0,Y 126.381,Z 482.711,A -85,B 0,C 180,E1 -25286.812,E2 -25286.812} C_VEL
LIN {X 0,Y 126.321,Z 483,A -85,B 0,C 180,E1 -25290,E2 -25290} C_VEL
LIN {X 0,Y 126.381,Z 482.7,A -85,B 0,C 180,E1 -25293.188,E2 -25293.188} C_VEL
LIN {X 0,Y 126.593,Z 481.91,A -85,B 0,C 180,E1 -25296.375,E2 -25296.375} C_VEL
LIN {X 0,Y 127.14,Z 480.65,A -85,B 0,C 180,E1 -25299.545,E2 -25299.545} C_VEL
LIN {X 0,Y 128.573,Z 477.745,A -85,B 0,C 180,E1 -25304.239,E2 -25304.239} C_VEL
LIN {X 0,Y 129.9,Z 475.095,A -85,B 0,C 180,E1 -25307.311,E2 -25307.311} C_VEL
LIN {X 0,Y 132.548,Z 469.918,A -85,B 0,C 180,E1 -25311.786,E2 -25311.786} C_VEL
LIN {X 0,Y 135.987,Z 463.084,A -85,B 0,C 180,E1 -25316.058,E2 -25316.058} C_VEL
LIN {X 0,Y 139.428,Z 455.618,A -85,B 0,C 180,E1 -25319.436,E2 -25319.436} C_VEL
LIN {X 0,Y 142.46,Z 448.251,A -85,B 0,C 180,E1 -25322.027,E2 -25322.027} C_VEL
LIN {X 0,Y 145.366,Z 440.357,A -85,B 0,C 180,E1 -25324.196,E2 -25324.196} C_VEL
LIN {X 0,Y 148.37,Z 430.625,A -85,B 0,C 180,E1 -25326.272,E2 -25326.272} C_VEL
LIN {X 0,Y 150.947,Z 419.921,A -85,B 0,C 180,E1 -25327.922,E2 -25327.922} C_VEL
LIN {X 0,Y 151.68,Z 414.381,A -85,B 0,C 180,E1 -25328.677,E2 -25328.677} C_VEL
LIN {X 0,Y 151.456,Z 408.909,A -85,B 0,C 180,E1 -25329.554,E2 -25329.554} C_VEL
LIN {X 0,Y 149.633,Z 396.029,A -85,B 0,C 180,E1 -25331.427,E2 -25331.427} C_VEL
LIN {X 0,Y 149.411,Z 390.234,A -85,B 0,C 180,E1 -25331.875,E2 -25331.875} C_VEL
LIN {X 0,Y 150.07,Z 378.013,A -85,B 0,C 180,E1 -25332.421,E2 -25332.421} C_VEL
LIN {X 0,Y 145.877,Z 366.867,A -85,B 0,C 180,E1 -25334.694,E2 -25334.694} C_VEL
LIN {X 0,Y 143.399,Z 361.62,A -85,B 0,C 180,E1 -25336.051,E2 -25336.051} C_VEL
LIN {X 0,Y 138.063,Z 352.799,A -85,B 0,C 180,E1 -25339.078,E2 -25339.078} C_VEL
LIN {X 0,Y 134.747,Z 347.949,A -85,B 0,C 180,E1 -25341.133,E2 -25341.133} C_VEL
LIN {X 0,Y 132.296,Z 344.461,A -85,B 0,C 180,E1 -25342.773,E2 -25342.773} C_VEL
LIN {X 0,Y 129.881,Z 340.918,A -85,B 0,C 180,E1 -25344.527,E2 -25344.527} C_VEL
LIN {X 0,Y 127.077,Z 337.719,A -85,B 0,C 180,E1 -25346.661,E2 -25346.661} C_VEL
LIN {X 0,Y 125.865,Z 335.617,A -85,B 0,C 180,E1 -25347.728,E2 -25347.728} C_VEL
LIN {X 0,Y 123.384,Z 333.541,A -85,B 0,C 180,E1 -25349.834,E2 -25349.834} C_VEL
LIN {X 0,Y 122.049,Z 330.719,A -85,B 0,C 180,E1 -25351.517,E2 -25351.517} C_VEL
LIN {X 0,Y 121.926,Z 330.117,A -85,B 0,C 180,E1 -25353.005,E2 -25353.005} C_VEL
LIN {X 0,Y 121.982,Z 330.07,A -85,B 0,C 180,E1 -25357.193,E2 -25357.193} C_VEL
LIN {X 0,Y 122.055,Z 330.076,A -85,B 0,C 180,E1 -25363.268,E2 -25363.268} C_VEL
LIN {X 0,Y 122.283,Z 330.031,A -85,B 0,C 180,E1 -25367.693,E2 -25367.693} C_VEL
LIN {X 0,Y 122.391,Z 330.047,A -85,B 0,C 180,E1 -25370.081,E2 -25370.081} C_VEL
LIN {X 0,Y 122.55,Z 329.996,A -85,B 0,C 180,E1 -25376.713,E2 -25376.713} C_VEL
LIN {X 0,Y 123.014,Z 329.976,A -85,B 0,C 180,E1 -25380,E2 -25380} C_VEL
LIN {X 0,Y 122.379,Z 330.02,A -85,B 0,C 180,E1 -25386.861,E2 -25386.861} C_VEL
LIN {X 0,Y 122.283,Z 330.032,A -85,B 0,C 180,E1 -25392.307,E2 -25392.307} C_VEL
LIN {X 0,Y 122.055,Z 330.075,A -85,B 0,C 180,E1 -25396.733,E2 -25396.733} C_VEL
LIN {X 0,Y 121.983,Z 330.07,A -85,B 0,C 180,E1 -25402.808,E2 -25402.808} C_VEL
LIN {X 0,Y 121.96,Z 330.396,A -85,B 0,C 180,E1 -25408.053,E2 -25408.053} C_VEL
LIN {X 0,Y 122.29,Z 331.466,A -85,B 0,C 180,E1 -25409.027,E2 -25409.027} C_VEL
LIN {X 0,Y 123.77,Z 333.98,A -85,B 0,C 180,E1 -25410.566,E2 -25410.566} C_VEL
LIN {X 0,Y 126.249,Z 336.037,A -85,B 0,C 180,E1 -25412.635,E2 -25412.635} C_VEL
LIN {X 0,Y 128.238,Z 339.302,A -85,B 0,C 180,E1 -25414.318,E2 -25414.318} C_VEL
LIN {X 0,Y 129.949,Z 341.013,A -85,B 0,C 180,E1 -25415.569,E2 -25415.569} C_VEL
LIN {X 0,Y 132.405,Z 344.578,A -85,B 0,C 180,E1 -25417.344,E2 -25417.344} C_VEL
LIN {X 0,Y 136.968,Z 351.249,A -85,B 0,C 180,E1 -25420.313,E2 -25420.313} C_VEL
LIN {X 0,Y 142.423,Z 359.901,A -85,B 0,C 180,E1 -25423.462,E2 -25423.462} C_VEL
LIN {X 0,Y 144.815,Z 364.433,A -85,B 0,C 180,E1 -25424.766,E2 -25424.766} C_VEL
LIN {X 0,Y 148.668,Z 374.017,A -85,B 0,C 180,E1 -25426.87,E2 -25426.87} C_VEL
LIN {X 0,Y 150.081,Z 378.049,A -85,B 0,C 180,E1 -25427.63,E2 -25427.63} C_VEL
LIN {X 0,Y 148.432,Z 401.707,A -85,B 0,C 180,E1 -25428.703,E2 -25428.703} C_VEL
LIN {X 0,Y 146.868,Z 412.685,A -85,B 0,C 180,E1 -25429.558,E2 -25429.558} C_VEL
LIN {X 0,Y 144.399,Z 424.274,A -85,B 0,C 180,E1 -25431.042,E2 -25431.042} C_VEL
LIN {X 0,Y 141.966,Z 433.197,A -85,B 0,C 180,E1 -25432.623,E2 -25432.623} C_VEL
LIN {X 0,Y 139.174,Z 441.459,A -85,B 0,C 180,E1 -25434.499,E2 -25434.499} C_VEL
LIN {X 0,Y 136.555,Z 448.144,A -85,B 0,C 180,E1 -25436.41,E2 -25436.41} C_VEL
LIN {X 0,Y 133.354,Z 455.528,A -85,B 0,C 180,E1 -25439.081,E2 -25439.081} C_VEL
LIN {X 0,Y 129.685,Z 463.011,A -85,B 0,C 180,E1 -25442.572,E2 -25442.572} C_VEL
LIN {X 0,Y 126.014,Z 469.866,A -85,B 0,C 180,E1 -25447.021,E2 -25447.021} C_VEL
LIN {X 0,Y 123.17,Z 475.054,A -85,B 0,C 180,E1 -25451.71,E2 -25451.71} C_VEL
LIN {X 0,Y 121.721,Z 477.714,A -85,B 0,C 180,E1 -25454.941,E2 -25454.941} C_VEL
LIN {X 0,Y 120.142,Z 480.628,A -85,B 0,C 180,E1 -25459.893,E2 -25459.893} C_VEL
LIN {X 0,Y 119.553,Z 481.897,A -85,B 0,C 180,E1 -25463.248,E2 -25463.248} C_VEL
LIN {X 0,Y 119.293,Z 482.695,A -85,B 0,C 180,E1 -25466.623,E2 -25466.623} C_VEL
LIN {X 0,Y 119.236,Z 482.999,A -85,B 0,C 180,E1 -25470,E2 -25470} C_VEL
LIN {X 0,Y 119.293,Z 482.716,A -85,B 0,C 180,E1 -25473.377,E2 -25473.377} C_VEL
LIN {X 0,Y 119.553,Z 481.958,A -85,B 0,C 180,E1 -25476.752,E2 -25476.752} C_VEL
LIN {X 0,Y 120.141,Z 480.731,A -85,B 0,C 180,E1 -25480.107,E2 -25480.107} C_VEL
LIN {X 0,Y 121.692,Z 477.859,A -85,B 0,C 180,E1 -25485.063,E2 -25485.063} C_VEL
LIN {X 0,Y 123.126,Z 475.245,A -85,B 0,C 180,E1 -25488.296,E2 -25488.296} C_VEL
LIN {X 0,Y 125.979,Z 470.109,A -85,B 0,C 180,E1 -25492.986,E2 -25492.986} C_VEL
LIN {X 0,Y 128.947,Z 464.584,A -85,B 0,C 180,E1 -25496.721,E2 -25496.721} C_VEL
LIN {X 0,Y 132.485,Z 457.638,A -85,B 0,C 180,E1 -25500.261,E2 -25500.261} C_VEL
LIN {X 0,Y 136.069,Z 449.667,A -85,B 0,C 180,E1 -25503.283,E2 -25503.283} C_VEL
LIN {X 0,Y 139.12,Z 442.067,A -85,B 0,C 180,E1 -25505.517,E2 -25505.517} C_VEL
LIN {X 0,Y 141.67,Z 434.594,A -85,B 0,C 180,E1 -25507.274,E2 -25507.274} C_VEL
LIN {X 0,Y 144.266,Z 425.612,A -85,B 0,C 180,E1 -25508.902,E2 -25508.902} C_VEL
LIN {X 0,Y 146.131,Z 417.036,A -85,B 0,C 180,E1 -25510.118,E2 -25510.118} C_VEL
LIN {X 0,Y 147.863,Z 407.441,A -85,B 0,C 180,E1 -25511.052,E2 -25511.052} C_VEL
LIN {X 0,Y 149.134,Z 395.759,A -85,B 0,C 180,E1 -25511.796,E2 -25511.796} C_VEL
LIN {X 0,Y 150.176,Z 378.038,A -85,B 0,C 180,E1 -25512.562,E2 -25512.562} C_VEL
LIN {X 0,Y 145.849,Z 366.592,A -85,B 0,C 180,E1 -25514.916,E2 -25514.916} C_VEL
LIN {X 0,Y 143.507,Z 361.74,A -85,B 0,C 180,E1 -25516.198,E2 -25516.198} C_VEL
LIN {X 0,Y 138.384,Z 353.182,A -85,B 0,C 180,E1 -25519.115,E2 -25519.115} C_VEL
LIN {X 0,Y 132.643,Z 344.812,A -85,B 0,C 180,E1 -25522.794,E2 -25522.794} C_VEL
LIN {X 0,Y 130.064,Z 341.207,A -85,B 0,C 180,E1 -25524.651,E2 -25524.651} C_VEL
LIN {X 0,Y 128.647,Z 339.707,A -85,B 0,C 180,E1 -25525.695,E2 -25525.695} C_VEL
LIN {X 0,Y 126.62,Z 336.856,A -85,B 0,C 180,E1 -25527.354,E2 -25527.354} C_VEL
LIN {X 0,Y 125.922,Z 335.654,A -85,B 0,C 180,E1 -25527.98,E2 -25527.98} C_VEL
LIN {X 0,Y 123.375,Z 333.516,A -85,B 0,C 180,E1 -25530.166,E2 -25530.166} C_VEL
LIN {X 0,Y 122.001,Z 330.656,A -85,B 0,C 180,E1 -25531.957,E2 -25531.957} C_VEL
LIN {X 0,Y 121.931,Z 330.115,A -85,B 0,C 180,E1 -25533.467,E2 -25533.467} C_VEL
LIN {X 0,Y 121.983,Z 330.071,A -85,B 0,C 180,E1 -25537.192,E2 -25537.192} C_VEL
LIN {X 0,Y 122.055,Z 330.077,A -85,B 0,C 180,E1 -25543.267,E2 -25543.267} C_VEL
LIN {X 0,Y 122.284,Z 330.031,A -85,B 0,C 180,E1 -25547.692,E2 -25547.692} C_VEL
LIN {X 0,Y 122.391,Z 330.046,A -85,B 0,C 180,E1 -25550.08,E2 -25550.08} C_VEL
LIN {X 0,Y 122.55,Z 329.996,A -85,B 0,C 180,E1 -25556.712,E2 -25556.712} C_VEL
LIN {X 0,Y 123.014,Z 329.975,A -85,B 0,C 180,E1 -25560,E2 -25560} C_VEL
LIN {X 0,Y 122.394,Z 330.019,A -85,B 0,C 180,E1 -25566.594,E2 -25566.594} C_VEL
LIN {X 0,Y 122.385,Z 330.047,A -85,B 0,C 180,E1 -25569.92,E2 -25569.92} C_VEL
LIN {X 0,Y 122.183,Z 330.04,A -85,B 0,C 180,E1 -25573.302,E2 -25573.302} C_VEL
LIN {X 0,Y 121.983,Z 330.078,A -85,B 0,C 180,E1 -25580.223,E2 -25580.223} C_VEL
LIN {X 0,Y 121.938,Z 330.103,A -85,B 0,C 180,E1 -25585.611,E2 -25585.611} C_VEL
LIN {X 0,Y 121.972,Z 330.419,A -85,B 0,C 180,E1 -25587.748,E2 -25587.748} C_VEL
LIN {X 0,Y 122.351,Z 331.699,A -85,B 0,C 180,E1 -25588.783,E2 -25588.783} C_VEL
LIN {X 0,Y 124.037,Z 334.28,A -85,B 0,C 180,E1 -25590.492,E2 -25590.492} C_VEL
LIN {X 0,Y 126.195,Z 335.968,A -85,B 0,C 180,E1 -25592.295,E2 -25592.295} C_VEL
LIN {X 0,Y 128.263,Z 339.327,A -85,B 0,C 180,E1 -25594.061,E2 -25594.061} C_VEL
LIN {X 0,Y 130.074,Z 341.24,A -85,B 0,C 180,E1 -25595.403,E2 -25595.403} C_VEL
LIN {X 0,Y 132.575,Z 344.716,A -85,B 0,C 180,E1 -25597.204,E2 -25597.204} C_VEL
LIN {X 0,Y 136.888,Z 351.084,A -85,B 0,C 180,E1 -25600.035,E2 -25600.035} C_VEL
LIN {X 0,Y 141.082,Z 357.539,A -85,B 0,C 180,E1 -25602.502,E2 -25602.502} C_VEL
LIN {X 0,Y 144.718,Z 364.079,A -85,B 0,C 180,E1 -25604.507,E2 -25604.507} C_VEL
LIN {X 0,Y 149.228,Z 375.222,A -85,B 0,C 180,E1 -25606.966,E2 -25606.966} C_VEL
LIN {X 0,Y 150.243,Z 378.203,A -85,B 0,C 180,E1 -25607.517,E2 -25607.517} C_VEL
LIN {X 0,Y 148.671,Z 401.219,A -85,B 0,C 180,E1 -25608.563,E2 -25608.563} C_VEL
LIN {X 0,Y 146.984,Z 413.053,A -85,B 0,C 180,E1 -25609.478,E2 -25609.478} C_VEL
LIN {X 0,Y 144.677,Z 423.796,A -85,B 0,C 180,E1 -25610.84,E2 -25610.84} C_VEL
LIN {X 0,Y 142.192,Z 432.777,A -85,B 0,C 180,E1 -25612.391,E2 -25612.391} C_VEL
LIN {X 0,Y 139.554,Z 440.713,A -85,B 0,C 180,E1 -25614.167,E2 -25614.167} C_VEL
LIN {X 0,Y 136.499,Z 448.542,A -85,B 0,C 180,E1 -25616.394,E2 -25616.394} C_VEL
LIN {X 0,Y 133.299,Z 455.864,A -85,B 0,C 180,E1 -25619.066,E2 -25619.066} C_VEL
LIN {X 0,Y 129.651,Z 463.288,A -85,B 0,C 180,E1 -25622.565,E2 -25622.565} C_VEL
LIN {X 0,Y 126.559,Z 469.103,A -85,B 0,C 180,E1 -25626.26,E2 -25626.26} C_VEL
LIN {X 0,Y 124.012,Z 473.688,A -85,B 0,C 180,E1 -25630.122,E2 -25630.122} C_VEL
LIN {X 0,Y 122.37,Z 476.668,A -85,B 0,C 180,E1 -25633.312,E2 -25633.312} C_VEL
LIN {X 0,Y 121.091,Z 478.98,A -85,B 0,C 180,E1 -25636.576,E2 -25636.576} C_VEL
LIN {X 0,Y 120.186,Z 480.709,A -85,B 0,C 180,E1 -25639.897,E2 -25639.897} C_VEL
LIN {X 0,Y 119.557,Z 481.946,A -85,B 0,C 180,E1 -25643.248,E2 -25643.248} C_VEL
LIN {X 0,Y 119.292,Z 482.711,A -85,B 0,C 180,E1 -25646.623,E2 -25646.623} C_VEL
LIN {X 0,Y 119.234,Z 483,A -85,B 0,C 180,E1 -25650,E2 -25650} C_VEL
LIN {X 0,Y 119.291,Z 482.699,A -85,B 0,C 180,E1 -25653.377,E2 -25653.377} C_VEL
LIN {X 0,Y 119.551,Z 481.91,A -85,B 0,C 180,E1 -25656.752,E2 -25656.752} C_VEL
LIN {X 0,Y 120.139,Z 480.649,A -85,B 0,C 180,E1 -25660.107,E2 -25660.107} C_VEL
LIN {X 0,Y 121.696,Z 477.744,A -85,B 0,C 180,E1 -25665.062,E2 -25665.062} C_VEL
LIN {X 0,Y 123.141,Z 475.094,A -85,B 0,C 180,E1 -25668.294,E2 -25668.294} C_VEL
LIN {X 0,Y 125.974,Z 469.916,A -85,B 0,C 180,E1 -25672.987,E2 -25672.987} C_VEL
LIN {X 0,Y 129.651,Z 463.082,A -85,B 0,C 180,E1 -25677.435,E2 -25677.435} C_VEL
LIN {X 0,Y 133.294,Z 455.615,A -85,B 0,C 180,E1 -25680.935,E2 -25680.935} C_VEL
LIN {X 0,Y 136.481,Z 448.248,A -85,B 0,C 180,E1 -25683.611,E2 -25683.611} C_VEL
LIN {X 0,Y 139.564,Z 440.353,A -85,B 0,C 180,E1 -25685.83,E2 -25685.83} C_VEL
LIN {X 0,Y 142.468,Z 431.396,A -85,B 0,C 180,E1 -25687.803,E2 -25687.803} C_VEL
LIN {X 0,Y 145.382,Z 420.103,A -85,B 0,C 180,E1 -25689.616,E2 -25689.616} C_VEL
LIN {X 0,Y 147.361,Z 409.67,A -85,B 0,C 180,E1 -25690.74,E2 -25690.74} C_VEL
LIN {X 0,Y 148.586,Z 400.792,A -85,B 0,C 180,E1 -25691.369,E2 -25691.369} C_VEL
LIN {X 0,Y 149.411,Z 390.234,A -85,B 0,C 180,E1 -25691.875,E2 -25691.875} C_VEL
LIN {X 0,Y 149.019,Z 386.491,A -85,B 0,C 180,E1 -25692.248,E2 -25692.248} C_VEL
LIN {X 0,Y 147.801,Z 383.12,A -85,B 0,C 180,E1 -25692.896,E2 -25692.896} C_VEL
LIN {X 0,Y 143.157,Z 375.019,A -85,B 0,C 180,E1 -25695.209,E2 -25695.209} C_VEL
LIN {X 0,Y 142.174,Z 372.816,A -85,B 0,C 180,E1 -25695.766,E2 -25695.766} C_VEL
LIN {X 0,Y 139.551,Z 366.699,A -85,B 0,C 180,E1 -25697.335,E2 -25697.335} C_VEL
LIN {X 0,Y 134.583,Z 358.181,A -85,B 0,C 180,E1 -25700.373,E2 -25700.373} C_VEL
LIN {X 0,Y 129.514,Z 350.5,A -85,B 0,C 180,E1 -25703.863,E2 -25703.863} C_VEL
LIN {X 0,Y 126.336,Z 346.136,A -85,B 0,C 180,E1 -25706.32,E2 -25706.32} C_VEL
LIN {X 0,Y 123.915,Z 342.833,A -85,B 0,C 180,E1 -25708.394,E2 -25708.394} C_VEL
LIN {X 0,Y 123.149,Z 341.766,A -85,B 0,C 180,E1 -25709.095,E2 -25709.095} C_VEL
LIN {X 0,Y 120.761,Z 339.311,A -85,B 0,C 180,E1 -25711.338,E2 -25711.338} C_VEL
LIN {X 0,Y 119.419,Z 336.768,A -85,B 0,C 180,E1 -25712.865,E2 -25712.865} C_VEL
LIN {X 0,Y 116.676,Z 334.855,A -85,B 0,C 180,E1 -25715.902,E2 -25715.902} C_VEL
LIN {X 0,Y 115.069,Z 331.782,A -85,B 0,C 180,E1 -25718.503,E2 -25718.503} C_VEL
LIN {X 0,Y 114.931,Z 331.026,A -85,B 0,C 180,E1 -25720.347,E2 -25720.347} C_VEL
LIN {X 0,Y 115.2,Z 330.911,A -85,B 0,C 180,E1 -25727.444,E2 -25727.444} C_VEL
LIN {X 0,Y 115.345,Z 330.899,A -85,B 0,C 180,E1 -25733.001,E2 -25733.001} C_VEL
LIN {X 0,Y 115.965,Z 330.853,A -85,B 0,C 180,E1 -25740,E2 -25740} C_VEL
LIN {X 0,Y 115.338,Z 330.899,A -85,B 0,C 180,E1 -25747,E2 -25747} C_VEL
LIN {X 0,Y 115.2,Z 330.911,A -85,B 0,C 180,E1 -25752.556,E2 -25752.556} C_VEL
LIN {X 0,Y 114.965,Z 331.079,A -85,B 0,C 180,E1 -25760.113,E2 -25760.113} C_VEL
LIN {X 0,Y 115.13,Z 332.022,A -85,B 0,C 180,E1 -25761.775,E2 -25761.775} C_VEL
LIN {X 0,Y 116.832,Z 335.061,A -85,B 0,C 180,E1 -25764.344,E2 -25764.344} C_VEL
LIN {X 0,Y 119.554,Z 337.032,A -85,B 0,C 180,E1 -25767.34,E2 -25767.34} C_VEL
LIN {X 0,Y 121.571,Z 340.374,A -85,B 0,C 180,E1 -25769.522,E2 -25769.522} C_VEL
LIN {X 0,Y 123.721,Z 342.422,A -85,B 0,C 180,E1 -25771.46,E2 -25771.46} C_VEL
LIN {X 0,Y 126.075,Z 345.877,A -85,B 0,C 180,E1 -25773.52,E2 -25773.52} C_VEL
LIN {X 0,Y 127.403,Z 347.541,A -85,B 0,C 180,E1 -25774.575,E2 -25774.575} C_VEL
LIN {X 0,Y 130.821,Z 352.496,A -85,B 0,C 180,E1 -25777.136,E2 -25777.136} C_VEL
LIN {X 0,Y 135.587,Z 359.879,A -85,B 0,C 180,E1 -25780.317,E2 -25780.317} C_VEL
LIN {X 0,Y 140.208,Z 367.922,A -85,B 0,C 180,E1 -25783.09,E2 -25783.09} C_VEL
LIN {X 0,Y 144.016,Z 377.795,A -85,B 0,C 180,E1 -25785.369,E2 -25785.369} C_VEL
LIN {X 0,Y 144.784,Z 380.129,A -85,B 0,C 180,E1 -25785.827,E2 -25785.827} C_VEL
LIN {X 0,Y 143.194,Z 401.724,A -85,B 0,C 180,E1 -25786.835,E2 -25786.835} C_VEL
LIN {X 0,Y 141.431,Z 413.375,A -85,B 0,C 180,E1 -25787.773,E2 -25787.773} C_VEL
LIN {X 0,Y 138.916,Z 424.442,A -85,B 0,C 180,E1 -25789.231,E2 -25789.231} C_VEL
LIN {X 0,Y 136.388,Z 433.195,A -85,B 0,C 180,E1 -25790.809,E2 -25790.809} C_VEL
LIN {X 0,Y 133.474,Z 441.463,A -85,B 0,C 180,E1 -25792.734,E2 -25792.734} C_VEL
LIN {X 0,Y 130.69,Z 448.147,A -85,B 0,C 180,E1 -25794.684,E2 -25794.684} C_VEL
LIN {X 0,Y 127.326,Z 455.531,A -85,B 0,C 180,E1 -25797.442,E2 -25797.442} C_VEL
LIN {X 0,Y 123.436,Z 463.013,A -85,B 0,C 180,E1 -25801.056,E2 -25801.056} C_VEL
LIN {X 0,Y 119.493,Z 469.868,A -85,B 0,C 180,E1 -25805.689,E2 -25805.689} C_VEL
LIN {X 0,Y 116.455,Z 475.055,A -85,B 0,C 180,E1 -25810.615,E2 -25810.615} C_VEL
LIN {X 0,Y 114.881,Z 477.715,A -85,B 0,C 180,E1 -25814.021,E2 -25814.021} C_VEL
LIN {X 0,Y 113.148,Z 480.629,A -85,B 0,C 180,E1 -25819.261,E2 -25819.261} C_VEL
LIN {X 0,Y 112.501,Z 481.897,A -85,B 0,C 180,E1 -25822.823,E2 -25822.823} C_VEL
LIN {X 0,Y 112.213,Z 482.695,A -85,B 0,C 180,E1 -25826.409,E2 -25826.409} C_VEL
LIN {X 0,Y 112.142,Z 482.999,A -85,B 0,C 180,E1 -25830,E2 -25830} C_VEL
LIN {X 0,Y 112.213,Z 482.715,A -85,B 0,C 180,E1 -25833.591,E2 -25833.591} C_VEL
LIN {X 0,Y 112.501,Z 481.958,A -85,B 0,C 180,E1 -25837.177,E2 -25837.177} C_VEL
LIN {X 0,Y 113.146,Z 480.73,A -85,B 0,C 180,E1 -25840.739,E2 -25840.739} C_VEL
LIN {X 0,Y 114.851,Z 477.858,A -85,B 0,C 180,E1 -25845.983,E2 -25845.983} C_VEL
LIN {X 0,Y 116.395,Z 475.243,A -85,B 0,C 180,E1 -25849.395,E2 -25849.395} C_VEL
LIN {X 0,Y 119.46,Z 470.107,A -85,B 0,C 180,E1 -25854.319,E2 -25854.319} C_VEL
LIN {X 0,Y 122.65,Z 464.582,A -85,B 0,C 180,E1 -25858.211,E2 -25858.211} C_VEL
LIN {X 0,Y 126.41,Z 457.636,A -85,B 0,C 180,E1 -25861.881,E2 -25861.881} C_VEL
LIN {X 0,Y 130.183,Z 449.663,A -85,B 0,C 180,E1 -25865,E2 -25865} C_VEL
LIN {X 0,Y 133.422,Z 442.063,A -85,B 0,C 180,E1 -25867.283,E2 -25867.283} C_VEL
LIN {X 0,Y 136.079,Z 434.589,A -85,B 0,C 180,E1 -25869.088,E2 -25869.088} C_VEL
LIN {X 0,Y 138.821,Z 425.605,A -85,B 0,C 180,E1 -25870.74,E2 -25870.74} C_VEL
LIN {X 0,Y 140.703,Z 417.445,A -85,B 0,C 180,E1 -25871.924,E2 -25871.924} C_VEL
LIN {X 0,Y 142.491,Z 408.113,A -85,B 0,C 180,E1 -25872.862,E2 -25872.862} C_VEL
LIN {X 0,Y 143.636,Z 398.519,A -85,B 0,C 180,E1 -25873.533,E2 -25873.533} C_VEL
LIN {X 0,Y 144.941,Z 380.138,A -85,B 0,C 180,E1 -25874.349,E2 -25874.349} C_VEL
LIN {X 0,Y 141.018,Z 369.615,A -85,B 0,C 180,E1 -25876.687,E2 -25876.687} C_VEL
LIN {X 0,Y 138.02,Z 363.804,A -85,B 0,C 180,E1 -25878.467,E2 -25878.467} C_VEL
LIN {X 0,Y 133.145,Z 355.917,A -85,B 0,C 180,E1 -25881.557,E2 -25881.557} C_VEL
LIN {X 0,Y 129.193,Z 350.078,A -85,B 0,C 180,E1 -25884.362,E2 -25884.362} C_VEL
LIN {X 0,Y 126.493,Z 346.258,A -85,B 0,C 180,E1 -25886.486,E2 -25886.486} C_VEL
LIN {X 0,Y 124.005,Z 342.95,A -85,B 0,C 180,E1 -25888.62,E2 -25888.62} C_VEL
LIN {X 0,Y 123.278,Z 341.866,A -85,B 0,C 180,E1 -25889.299,E2 -25889.299} C_VEL
LIN {X 0,Y 120.794,Z 339.34,A -85,B 0,C 180,E1 -25891.652,E2 -25891.652} C_VEL
LIN {X 0,Y 119.336,Z 336.729,A -85,B 0,C 180,E1 -25893.317,E2 -25893.317} C_VEL
LIN {X 0,Y 116.773,Z 334.947,A -85,B 0,C 180,E1 -25896.201,E2 -25896.201} C_VEL
LIN {X 0,Y 115.171,Z 332.151,A -85,B 0,C 180,E1 -25898.639,E2 -25898.639} C_VEL
LIN {X 0,Y 114.986,Z 331.228,A -85,B 0,C 180,E1 -25899.891,E2 -25899.891} C_VEL
LIN {X 0,Y 115.201,Z 330.911,A -85,B 0,C 180,E1 -25907.443,E2 -25907.443} C_VEL
LIN {X 0,Y 115.345,Z 330.899,A -85,B 0,C 180,E1 -25913,E2 -25913} C_VEL
LIN {X 0,Y 115.965,Z 330.853,A -85,B 0,C 180,E1 -25920,E2 -25920} C_VEL
LIN {X 0,Y 115.338,Z 330.9,A -85,B 0,C 180,E1 -25927,E2 -25927} C_VEL
LIN {X 0,Y 115.2,Z 330.911,A -85,B 0,C 180,E1 -25932.555,E2 -25932.555} C_VEL
LIN {X 0,Y 114.97,Z 331.219,A -85,B 0,C 180,E1 -25940.111,E2 -25940.111} C_VEL
LIN {X 0,Y 115.233,Z 332.365,A -85,B 0,C 180,E1 -25941.561,E2 -25941.561} C_VEL
LIN {X 0,Y 117.12,Z 335.309,A -85,B 0,C 180,E1 -25944.279,E2 -25944.279} C_VEL
LIN {X 0,Y 119.561,Z 337.04,A -85,B 0,C 180,E1 -25946.982,E2 -25946.982} C_VEL
LIN {X 0,Y 121.472,Z 340.244,A -85,B 0,C 180,E1 -25949.088,E2 -25949.088} C_VEL
LIN {X 0,Y 123.734,Z 342.397,A -85,B 0,C 180,E1 -25951.158,E2 -25951.158} C_VEL
LIN {X 0,Y 126.086,Z 345.885,A -85,B 0,C 180,E1 -25953.241,E2 -25953.241} C_VEL
LIN {X 0,Y 127.429,Z 347.539,A -85,B 0,C 180,E1 -25954.315,E2 -25954.315} C_VEL
LIN {X 0,Y 130.94,Z 352.65,A -85,B 0,C 180,E1 -25956.966,E2 -25956.966} C_VEL
LIN {X 0,Y 135.936,Z 360.292,A -85,B 0,C 180,E1 -25960.297,E2 -25960.297} C_VEL
LIN {X 0,Y 140.411,Z 368.282,A -85,B 0,C 180,E1 -25962.997,E2 -25962.997} C_VEL
LIN {X 0,Y 144.511,Z 378.796,A -85,B 0,C 180,E1 -25965.438,E2 -25965.438} C_VEL
LIN {X 0,Y 144.956,Z 380.191,A -85,B 0,C 180,E1 -25965.706,E2 -25965.706} C_VEL
LIN {X 0,Y 143.425,Z 401.235,A -85,B 0,C 180,E1 -25966.686,E2 -25966.686} C_VEL
LIN {X 0,Y 141.638,Z 413.237,A -85,B 0,C 180,E1 -25967.634,E2 -25967.634} C_VEL
LIN {X 0,Y 139.239,Z 423.802,A -85,B 0,C 180,E1 -25968.993,E2 -25968.993} C_VEL
LIN {X 0,Y 136.771,Z 432.411,A -85,B 0,C 180,E1 -25970.503,E2 -25970.503} C_VEL
LIN {X 0,Y 133.874,Z 440.717,A -85,B 0,C 180,E1 -25972.391,E2 -25972.391} C_VEL
LIN {X 0,Y 130.631,Z 448.545,A -85,B 0,C 180,E1 -25974.666,E2 -25974.666} C_VEL
LIN {X 0,Y 127.265,Z 455.866,A -85,B 0,C 180,E1 -25977.424,E2 -25977.424} C_VEL
LIN {X 0,Y 123.401,Z 463.29,A -85,B 0,C 180,E1 -25981.048,E2 -25981.048} C_VEL
LIN {X 0,Y 120.083,Z 469.105,A -85,B 0,C 180,E1 -25984.893,E2 -25984.893} C_VEL
LIN {X 0,Y 117.366,Z 473.689,A -85,B 0,C 180,E1 -25988.944,E2 -25988.944} C_VEL
LIN {X 0,Y 115.586,Z 476.669,A -85,B 0,C 180,E1 -25992.301,E2 -25992.301} C_VEL
LIN {X 0,Y 114.201,Z 478.981,A -85,B 0,C 180,E1 -25995.75,E2 -25995.75} C_VEL
LIN {X 0,Y 113.2,Z 480.71,A -85,B 0,C 180,E1 -25999.266,E2 -25999.266} C_VEL
LIN {X 0,Y 112.506,Z 481.946,A -85,B 0,C 180,E1 -26002.823,E2 -26002.823} C_VEL
LIN {X 0,Y 112.212,Z 482.711,A -85,B 0,C 180,E1 -26006.409,E2 -26006.409} C_VEL
LIN {X 0,Y 112.14,Z 483,A -85,B 0,C 180,E1 -26010,E2 -26010} C_VEL
LIN {X 0,Y 112.211,Z 482.699,A -85,B 0,C 180,E1 -26013.591,E2 -26013.591} C_VEL
LIN {X 0,Y 112.499,Z 481.909,A -85,B 0,C 180,E1 -26017.177,E2 -26017.177} C_VEL
LIN {X 0,Y 113.145,Z 480.649,A -85,B 0,C 180,E1 -26020.739,E2 -26020.739} C_VEL
LIN {X 0,Y 114.855,Z 477.743,A -85,B 0,C 180,E1 -26025.983,E2 -26025.983} C_VEL
LIN {X 0,Y 116.407,Z 475.093,A -85,B 0,C 180,E1 -26029.393,E2 -26029.393} C_VEL
LIN {X 0,Y 119.458,Z 469.915,A -85,B 0,C 180,E1 -26034.319,E2 -26034.319} C_VEL
LIN {X 0,Y 123.401,Z 463.08,A -85,B 0,C 180,E1 -26038.952,E2 -26038.952} C_VEL
LIN {X 0,Y 127.259,Z 455.612,A -85,B 0,C 180,E1 -26042.578,E2 -26042.578} C_VEL
LIN {X 0,Y 130.204,Z 449.266,A -85,B 0,C 180,E1 -26044.994,E2 -26044.994} C_VEL
LIN {X 0,Y 133.407,Z 441.579,A -85,B 0,C 180,E1 -26047.287,E2 -26047.287} C_VEL
LIN {X 0,Y 136.186,Z 433.695,A -85,B 0,C 180,E1 -26049.147,E2 -26049.147} C_VEL
LIN {X 0,Y 138.35,Z 426.436,A -85,B 0,C 180,E1 -26050.505,E2 -26050.505} C_VEL
LIN {X 0,Y 140.316,Z 418.631,A -85,B 0,C 180,E1 -26051.64,E2 -26051.64} C_VEL
LIN {X 0,Y 142.159,Z 408.985,A -85,B 0,C 180,E1 -26052.669,E2 -26052.669} C_VEL
LIN {X 0,Y 143.424,Z 399.665,A -85,B 0,C 180,E1 -26053.315,E2 -26053.315} C_VEL
LIN {X 0,Y 144.775,Z 379.947,A -85,B 0,C 180,E1 -26054.234,E2 -26054.234} C_VEL
LIN {X 0,Y 142.174,Z 372.816,A -85,B 0,C 180,E1 -26055.766,E2 -26055.766} C_VEL
LIN {X 0,Y 140.682,Z 369.859,A -85,B 0,C 180,E1 -26056.607,E2 -26056.607} C_VEL
LIN {X 0,Y 137.793,Z 366.352,A -85,B 0,C 180,E1 -26058.16,E2 -26058.16} C_VEL
LIN {X 0,Y 128.236,Z 358.429,A -85,B 0,C 180,E1 -26063.908,E2 -26063.908} C_VEL
LIN {X 0,Y 126.498,Z 356.194,A -85,B 0,C 180,E1 -26065.219,E2 -26065.219} C_VEL
LIN {X 0,Y 123.473,Z 351.92,A -85,B 0,C 180,E1 -26067.746,E2 -26067.746} C_VEL
LIN {X 0,Y 120.662,Z 347.956,A -85,B 0,C 180,E1 -26070.389,E2 -26070.389} C_VEL
LIN {X 0,Y 118.21,Z 345.073,A -85,B 0,C 180,E1 -26072.925,E2 -26072.925} C_VEL
LIN {X 0,Y 117.071,Z 343.191,A -85,B 0,C 180,E1 -26074.295,E2 -26074.295} C_VEL
LIN {X 0,Y 114.5,Z 340.894,A -85,B 0,C 180,E1 -26077.474,E2 -26077.474} C_VEL
LIN {X 0,Y 112.945,Z 337.942,A -85,B 0,C 180,E1 -26079.987,E2 -26079.987} C_VEL
LIN {X 0,Y 109.846,Z 335.763,A -85,B 0,C 180,E1 -26085.586,E2 -26085.586} C_VEL
LIN {X 0,Y 108.392,Z 332.587,A -85,B 0,C 180,E1 -26090.672,E2 -26090.672} C_VEL
LIN {X 0,Y 108.351,Z 331.852,A -85,B 0,C 180,E1 -26095.35,E2 -26095.35} C_VEL
LIN {X 0,Y 108.891,Z 331.741,A -85,B 0,C 180,E1 -26100,E2 -26100} C_VEL
LIN {X 0,Y 108.321,Z 332.097,A -85,B 0,C 180,E1 -26107.456,E2 -26107.456} C_VEL
LIN {X 0,Y 108.555,Z 333.138,A -85,B 0,C 180,E1 -26110.492,E2 -26110.492} C_VEL
LIN {X 0,Y 110.301,Z 336.283,A -85,B 0,C 180,E1 -26115.475,E2 -26115.475} C_VEL
LIN {X 0,Y 113.113,Z 338.214,A -85,B 0,C 180,E1 -26120.338,E2 -26120.338} C_VEL
LIN {X 0,Y 114.958,Z 341.513,A -85,B 0,C 180,E1 -26123.211,E2 -26123.211} C_VEL
LIN {X 0,Y 117.517,Z 343.745,A -85,B 0,C 180,E1 -26126.273,E2 -26126.273} C_VEL
LIN {X 0,Y 119.627,Z 346.958,A -85,B 0,C 180,E1 -26128.65,E2 -26128.65} C_VEL
LIN {X 0,Y 121.355,Z 348.864,A -85,B 0,C 180,E1 -26130.331,E2 -26130.331} C_VEL
LIN {X 0,Y 123.853,Z 352.341,A -85,B 0,C 180,E1 -26132.621,E2 -26132.621} C_VEL
LIN {X 0,Y 127.737,Z 358.156,A -85,B 0,C 180,E1 -26135.804,E2 -26135.804} C_VEL
LIN {X 0,Y 133.116,Z 366.857,A -85,B 0,C 180,E1 -26139.628,E2 -26139.628} C_VEL
LIN {X 0,Y 136.482,Z 373.344,A -85,B 0,C 180,E1 -26141.811,E2 -26141.811} C_VEL
LIN {X 0,Y 139.668,Z 382.192,A -85,B 0,C 180,E1 -26143.9,E2 -26143.9} C_VEL
LIN {X 0,Y 138.114,Z 401.741,A -85,B 0,C 180,E1 -26144.825,E2 -26144.825} C_VEL
LIN {X 0,Y 136.104,Z 414.127,A -85,B 0,C 180,E1 -26145.858,E2 -26145.858} C_VEL
LIN {X 0,Y 133.577,Z 424.611,A -85,B 0,C 180,E1 -26147.27,E2 -26147.27} C_VEL
LIN {X 0,Y 130.951,Z 433.198,A -85,B 0,C 180,E1 -26148.84,E2 -26148.84} C_VEL
LIN {X 0,Y 127.91,Z 441.467,A -85,B 0,C 180,E1 -26150.813,E2 -26150.813} C_VEL
LIN {X 0,Y 124.953,Z 448.151,A -85,B 0,C 180,E1 -26152.798,E2 -26152.798} C_VEL
LIN {X 0,Y 121.408,Z 455.534,A -85,B 0,C 180,E1 -26155.64,E2 -26155.64} C_VEL
LIN {X 0,Y 117.285,Z 463.015,A -85,B 0,C 180,E1 -26159.381,E2 -26159.381} C_VEL
LIN {X 0,Y 113.045,Z 469.87,A -85,B 0,C 180,E1 -26164.203,E2 -26164.203} C_VEL
LIN {X 0,Y 109.773,Z 475.057,A -85,B 0,C 180,E1 -26169.383,E2 -26169.383} C_VEL
LIN {X 0,Y 108.064,Z 477.716,A -85,B 0,C 180,E1 -26172.983,E2 -26172.983} C_VEL
LIN {X 0,Y 106.183,Z 480.629,A -85,B 0,C 180,E1 -26178.547,E2 -26178.547} C_VEL
LIN {X 0,Y 105.473,Z 481.898,A -85,B 0,C 180,E1 -26182.342,E2 -26182.342} C_VEL
LIN {X 0,Y 105.126,Z 482.695,A -85,B 0,C 180,E1 -26186.167,E2 -26186.167} C_VEL
LIN {X 0,Y 105.042,Z 482.999,A -85,B 0,C 180,E1 -26190,E2 -26190} C_VEL
LIN {X 0,Y 105.126,Z 482.715,A -85,B 0,C 180,E1 -26193.833,E2 -26193.833} C_VEL
LIN {X 0,Y 105.473,Z 481.958,A -85,B 0,C 180,E1 -26197.658,E2 -26197.658} C_VEL
LIN {X 0,Y 106.181,Z 480.729,A -85,B 0,C 180,E1 -26201.453,E2 -26201.453} C_VEL
LIN {X 0,Y 108.033,Z 477.857,A -85,B 0,C 180,E1 -26207.022,E2 -26207.022} C_VEL
LIN {X 0,Y 109.722,Z 475.242,A -85,B 0,C 180,E1 -26210.627,E2 -26210.627} C_VEL
LIN {X 0,Y 113.013,Z 470.105,A -85,B 0,C 180,E1 -26215.804,E2 -26215.804} C_VEL
LIN {X 0,Y 116.451,Z 464.58,A -85,B 0,C 180,E1 -26219.86,E2 -26219.86} C_VEL
LIN {X 0,Y 120.449,Z 457.633,A -85,B 0,C 180,E1 -26223.662,E2 -26223.662} C_VEL
LIN {X 0,Y 124.42,Z 449.66,A -85,B 0,C 180,E1 -26226.881,E2 -26226.881} C_VEL
LIN {X 0,Y 127.853,Z 442.059,A -85,B 0,C 180,E1 -26229.208,E2 -26229.208} C_VEL
LIN {X 0,Y 130.934,Z 433.73,A -85,B 0,C 180,E1 -26231.232,E2 -26231.232} C_VEL
LIN {X 0,Y 133.468,Z 425.772,A -85,B 0,C 180,E1 -26232.703,E2 -26232.703} C_VEL
LIN {X 0,Y 135.395,Z 417.918,A -85,B 0,C 180,E1 -26233.872,E2 -26233.872} C_VEL
LIN {X 0,Y 137.252,Z 408.802,A -85,B 0,C 180,E1 -26234.818,E2 -26234.818} C_VEL
LIN {X 0,Y 138.451,Z 399.763,A -85,B 0,C 180,E1 -26235.481,E2 -26235.481} C_VEL
LIN {X 0,Y 139.852,Z 382.268,A -85,B 0,C 180,E1 -26236.267,E2 -26236.267} C_VEL
LIN {X 0,Y 136.558,Z 373.341,A -85,B 0,C 180,E1 -26238.418,E2 -26238.418} C_VEL
LIN {X 0,Y 132.455,Z 365.572,A -85,B 0,C 180,E1 -26241.11,E2 -26241.11} C_VEL
LIN {X 0,Y 126.806,Z 356.522,A -85,B 0,C 180,E1 -26245.262,E2 -26245.262} C_VEL
LIN {X 0,Y 123.525,Z 351.968,A -85,B 0,C 180,E1 -26248.005,E2 -26248.005} C_VEL
LIN {X 0,Y 120.817,Z 348.029,A -85,B 0,C 180,E1 -26250.585,E2 -26250.585} C_VEL
LIN {X 0,Y 118.345,Z 345.228,A -85,B 0,C 180,E1 -26253.146,E2 -26253.146} C_VEL
LIN {X 0,Y 117.081,Z 343.192,A -85,B 0,C 180,E1 -26254.678,E2 -26254.678} C_VEL
LIN {X 0,Y 114.504,Z 340.855,A -85,B 0,C 180,E1 -26257.933,E2 -26257.933} C_VEL
LIN {X 0,Y 112.977,Z 337.925,A -85,B 0,C 180,E1 -26260.466,E2 -26260.466} C_VEL
LIN {X 0,Y 109.983,Z 335.864,A -85,B 0,C 180,E1 -26266.015,E2 -26266.015} C_VEL
LIN {X 0,Y 108.389,Z 332.522,A -85,B 0,C 180,E1 -26272.08,E2 -26272.08} C_VEL
LIN {X 0,Y 108.598,Z 331.794,A -85,B 0,C 180,E1 -26278.145,E2 -26278.145} C_VEL
LIN {X 0,Y 108.915,Z 331.754,A -85,B 0,C 180,E1 -26280,E2 -26280} C_VEL
LIN {X 0,Y 108.379,Z 332.346,A -85,B 0,C 180,E1 -26287.451,E2 -26287.451} C_VEL
LIN {X 0,Y 108.965,Z 334.215,A -85,B 0,C 180,E1 -26291.156,E2 -26291.156} C_VEL
LIN {X 0,Y 111.158,Z 336.964,A -85,B 0,C 180,E1 -26296.529,E2 -26296.529} C_VEL
LIN {X 0,Y 113.136,Z 338.218,A -85,B 0,C 180,E1 -26299.859,E2 -26299.859} C_VEL
LIN {X 0,Y 115.054,Z 341.564,A -85,B 0,C 180,E1 -26302.889,E2 -26302.889} C_VEL
LIN {X 0,Y 117.534,Z 343.706,A -85,B 0,C 180,E1 -26305.899,E2 -26305.899} C_VEL
LIN {X 0,Y 119.69,Z 347.008,A -85,B 0,C 180,E1 -26308.363,E2 -26308.363} C_VEL
LIN {X 0,Y 121.327,Z 348.771,A -85,B 0,C 180,E1 -26309.97,E2 -26309.97} C_VEL
LIN {X 0,Y 124.118,Z 352.605,A -85,B 0,C 180,E1 -26312.542,E2 -26312.542} C_VEL
LIN {X 0,Y 129.204,Z 360.253,A -85,B 0,C 180,E1 -26316.629,E2 -26316.629} C_VEL
LIN {X 0,Y 134.121,Z 368.561,A -85,B 0,C 180,E1 -26320.052,E2 -26320.052} C_VEL
LIN {X 0,Y 136.715,Z 373.681,A -85,B 0,C 180,E1 -26321.727,E2 -26321.727} C_VEL
LIN {X 0,Y 139.829,Z 382.159,A -85,B 0,C 180,E1 -26323.76,E2 -26323.76} C_VEL
LIN {X 0,Y 138.351,Z 401.251,A -85,B 0,C 180,E1 -26324.671,E2 -26324.671} C_VEL
LIN {X 0,Y 136.489,Z 413.199,A -85,B 0,C 180,E1 -26325.621,E2 -26325.621} C_VEL
LIN {X 0,Y 133.963,Z 423.807,A -85,B 0,C 180,E1 -26327,E2 -26327} C_VEL
LIN {X 0,Y 131.518,Z 431.94,A -85,B 0,C 180,E1 -26328.428,E2 -26328.428} C_VEL
LIN {X 0,Y 128.834,Z 439.492,A -85,B 0,C 180,E1 -26330.137,E2 -26330.137} C_VEL
LIN {X 0,Y 125.402,Z 447.528,A -85,B 0,C 180,E1 -26332.45,E2 -26332.45} C_VEL
LIN {X 0,Y 122.192,Z 454.165,A -85,B 0,C 180,E1 -26334.89,E2 -26334.89} C_VEL
LIN {X 0,Y 118.806,Z 460.466,A -85,B 0,C 180,E1 -26337.833,E2 -26337.833} C_VEL
LIN {X 0,Y 115.741,Z 465.7,A -85,B 0,C 180,E1 -26340.938,E2 -26340.938} C_VEL
LIN {X 0,Y 113.023,Z 470.062,A -85,B 0,C 180,E1 -26344.198,E2 -26344.198} C_VEL
LIN {X 0,Y 109.74,Z 475.207,A -85,B 0,C 180,E1 -26349.377,E2 -26349.377} C_VEL
LIN {X 0,Y 107.316,Z 478.982,A -85,B 0,C 180,E1 -26354.814,E2 -26354.814} C_VEL
LIN {X 0,Y 106.223,Z 480.711,A -85,B 0,C 180,E1 -26358.552,E2 -26358.552} C_VEL
LIN {X 0,Y 105.479,Z 481.946,A -85,B 0,C 180,E1 -26362.342,E2 -26362.342} C_VEL
LIN {X 0,Y 105.125,Z 482.712,A -85,B 0,C 180,E1 -26366.167,E2 -26366.167} C_VEL
LIN {X 0,Y 105.04,Z 483,A -85,B 0,C 180,E1 -26370,E2 -26370} C_VEL
LIN {X 0,Y 105.125,Z 482.699,A -85,B 0,C 180,E1 -26373.833,E2 -26373.833} C_VEL
LIN {X 0,Y 105.471,Z 481.909,A -85,B 0,C 180,E1 -26377.658,E2 -26377.658} C_VEL
LIN {X 0,Y 106.18,Z 480.648,A -85,B 0,C 180,E1 -26381.453,E2 -26381.453} C_VEL
LIN {X 0,Y 108.037,Z 477.742,A -85,B 0,C 180,E1 -26387.021,E2 -26387.021} C_VEL
LIN {X 0,Y 109.732,Z 475.092,A -85,B 0,C 180,E1 -26390.625,E2 -26390.625} C_VEL
LIN {X 0,Y 113.014,Z 469.913,A -85,B 0,C 180,E1 -26395.804,E2 -26395.804} C_VEL
LIN {X 0,Y 117.25,Z 463.078,A -85,B 0,C 180,E1 -26400.629,E2 -26400.629} C_VEL
LIN {X 0,Y 121.339,Z 455.61,A -85,B 0,C 180,E1 -26404.382,E2 -26404.382} C_VEL
LIN {X 0,Y 124.44,Z 449.262,A -85,B 0,C 180,E1 -26406.874,E2 -26406.874} C_VEL
LIN {X 0,Y 127.845,Z 441.576,A -85,B 0,C 180,E1 -26409.21,E2 -26409.21} C_VEL
LIN {X 0,Y 130.97,Z 433.084,A -85,B 0,C 180,E1 -26411.236,E2 -26411.236} C_VEL
LIN {X 0,Y 133.424,Z 425.021,A -85,B 0,C 180,E1 -26412.723,E2 -26412.723} C_VEL
LIN {X 0,Y 135.738,Z 415.799,A -85,B 0,C 180,E1 -26413.98,E2 -26413.98} C_VEL
LIN {X 0,Y 137.872,Z 403.978,A -85,B 0,C 180,E1 -26415.086,E2 -26415.086} C_VEL
LIN {X 0,Y 139.355,Z 387.489,A -85,B 0,C 180,E1 -26415.894,E2 -26415.894} C_VEL
LIN {X 0,Y 139.647,Z 381.988,A -85,B 0,C 180,E1 -26416.169,E2 -26416.169} C_VEL
LIN {X 0,Y 135.853,Z 371.893,A -85,B 0,C 180,E1 -26418.645,E2 -26418.645} C_VEL
LIN {X 0,Y 131.19,Z 363.58,A -85,B 0,C 180,E1 -26421.727,E2 -26421.727} C_VEL
LIN {X 0,Y 126.498,Z 356.194,A -85,B 0,C 180,E1 -26425.219,E2 -26425.219} C_VEL
LIN {X 0,Y 124.656,Z 354.533,A -85,B 0,C 180,E1 -26426.625,E2 -26426.625} C_VEL
LIN {X 0,Y 121.147,Z 353.872,A -85,B 0,C 180,E1 -26429.309,E2 -26429.309} C_VEL
LIN {X 0,Y 117.874,Z 353.322,A -85,B 0,C 180,E1 -26432.173,E2 -26432.173} C_VEL
LIN {X 0,Y 116.358,Z 351.808,A -85,B 0,C 180,E1 -26433.827,E2 -26433.827} C_VEL
LIN {X 0,Y 115.019,Z 349.66,A -85,B 0,C 180,E1 -26435.532,E2 -26435.532} C_VEL
LIN {X 0,Y 112.514,Z 347.056,A -85,B 0,C 180,E1 -26438.952,E2 -26438.952} C_VEL
LIN {X 0,Y 111.228,Z 344.575,A -85,B 0,C 180,E1 -26441.225,E2 -26441.225} C_VEL
LIN {X 0,Y 108.592,Z 342.572,A -85,B 0,C 180,E1 -26446.41,E2 -26446.41} C_VEL
LIN {X 0,Y 107.109,Z 339.415,A -85,B 0,C 180,E1 -26451.511,E2 -26451.511} C_VEL
LIN {X 0,Y 106.111,Z 338.418,A -85,B 0,C 180,E1 -26458.103,E2 -26458.103} C_VEL
LIN {X 0,Y 106.106,Z 338.434,A -85,B 0,C 180,E1 -26461.898,E2 -26461.898} C_VEL
LIN {X 0,Y 106.991,Z 339.25,A -85,B 0,C 180,E1 -26468.024,E2 -26468.024} C_VEL
LIN {X 0,Y 107.791,Z 341.141,A -85,B 0,C 180,E1 -26471.28,E2 -26471.28} C_VEL
LIN {X 0,Y 109.675,Z 343.686,A -85,B 0,C 180,E1 -26476.063,E2 -26476.063} C_VEL
LIN {X 0,Y 111.45,Z 344.891,A -85,B 0,C 180,E1 -26479.214,E2 -26479.214} C_VEL
LIN {X 0,Y 113.318,Z 348.185,A -85,B 0,C 180,E1 -26482.31,E2 -26482.31} C_VEL
LIN {X 0,Y 115.498,Z 350.299,A -85,B 0,C 180,E1 -26485.122,E2 -26485.122} C_VEL
LIN {X 0,Y 117.934,Z 353.807,A -85,B 0,C 180,E1 -26487.989,E2 -26487.989} C_VEL
LIN {X 0,Y 118.991,Z 355.164,A -85,B 0,C 180,E1 -26489.099,E2 -26489.099} C_VEL
LIN {X 0,Y 122.106,Z 359.768,A -85,B 0,C 180,E1 -26492.131,E2 -26492.131} C_VEL
LIN {X 0,Y 126.021,Z 365.842,A -85,B 0,C 180,E1 -26495.453,E2 -26495.453} C_VEL
LIN {X 0,Y 131.165,Z 375.001,A -85,B 0,C 180,E1 -26499.282,E2 -26499.282} C_VEL
LIN {X 0,Y 133.011,Z 379.177,A -85,B 0,C 180,E1 -26500.586,E2 -26500.586} C_VEL
LIN {X 0,Y 134.663,Z 384.177,A -85,B 0,C 180,E1 -26501.794,E2 -26501.794} C_VEL
LIN {X 0,Y 133.202,Z 401.758,A -85,B 0,C 180,E1 -26502.657,E2 -26502.657} C_VEL
LIN {X 0,Y 131.384,Z 412.898,A -85,B 0,C 180,E1 -26503.557,E2 -26503.557} C_VEL
LIN {X 0,Y 128.909,Z 423.074,A -85,B 0,C 180,E1 -26504.868,E2 -26504.868} C_VEL
LIN {X 0,Y 125.933,Z 432.556,A -85,B 0,C 180,E1 -26506.576,E2 -26506.576} C_VEL
LIN {X 0,Y 123.031,Z 440.241,A -85,B 0,C 180,E1 -26508.39,E2 -26508.39} C_VEL
LIN {X 0,Y 119.361,Z 448.154,A -85,B 0,C 180,E1 -26510.732,E2 -26510.732} C_VEL
LIN {X 0,Y 115.619,Z 455.536,A -85,B 0,C 180,E1 -26513.655,E2 -26513.655} C_VEL
LIN {X 0,Y 111.246,Z 463.017,A -85,B 0,C 180,E1 -26517.522,E2 -26517.522} C_VEL
LIN {X 0,Y 106.686,Z 469.871,A -85,B 0,C 180,E1 -26522.541,E2 -26522.541} C_VEL
LIN {X 0,Y 103.154,Z 475.058,A -85,B 0,C 180,E1 -26527.994,E2 -26527.994} C_VEL
LIN {X 0,Y 101.278,Z 477.717,A -85,B 0,C 180,E1 -26531.804,E2 -26531.804} C_VEL
LIN {X 0,Y 99.247,Z 480.63,A -85,B 0,C 180,E1 -26537.735,E2 -26537.735} C_VEL
LIN {X 0,Y 98.427,Z 481.898,A -85,B 0,C 180,E1 -26541.79,E2 -26541.79} C_VEL
LIN {X 0,Y 98.041,Z 482.696,A -85,B 0,C 180,E1 -26545.889,E2 -26545.889} C_VEL
LIN {X 0,Y 97.969,Z 482.999,A -85,B 0,C 180,E1 -26550,E2 -26550} C_VEL
LIN {X 0,Y 98.041,Z 482.715,A -85,B 0,C 180,E1 -26554.111,E2 -26554.111} C_VEL
LIN {X 0,Y 98.426,Z 481.957,A -85,B 0,C 180,E1 -26558.21,E2 -26558.21} C_VEL
LIN {X 0,Y 99.244,Z 480.729,A -85,B 0,C 180,E1 -26562.265,E2 -26562.265} C_VEL
LIN {X 0,Y 101.245,Z 477.856,A -85,B 0,C 180,E1 -26568.202,E2 -26568.202} C_VEL
LIN {X 0,Y 103.093,Z 475.241,A -85,B 0,C 180,E1 -26572.02,E2 -26572.02} C_VEL
LIN {X 0,Y 106.655,Z 470.104,A -85,B 0,C 180,E1 -26577.468,E2 -26577.468} C_VEL
LIN {X 0,Y 110.362,Z 464.578,A -85,B 0,C 180,E1 -26581.692,E2 -26581.692} C_VEL
LIN {X 0,Y 114.616,Z 457.631,A -85,B 0,C 180,E1 -26585.627,E2 -26585.627} C_VEL
LIN {X 0,Y 118.821,Z 449.657,A -85,B 0,C 180,E1 -26588.934,E2 -26588.934} C_VEL
LIN {X 0,Y 122.439,Z 442.055,A -85,B 0,C 180,E1 -26591.306,E2 -26591.306} C_VEL
LIN {X 0,Y 125.094,Z 435.404,A -85,B 0,C 180,E1 -26593.002,E2 -26593.002} C_VEL
LIN {X 0,Y 127.797,Z 427.715,A -85,B 0,C 180,E1 -26594.518,E2 -26594.518} C_VEL
LIN {X 0,Y 130.269,Z 418.394,A -85,B 0,C 180,E1 -26595.97,E2 -26595.97} C_VEL
LIN {X 0,Y 132.194,Z 409.491,A -85,B 0,C 180,E1 -26596.923,E2 -26596.923} C_VEL
LIN {X 0,Y 133.532,Z 400.174,A -85,B 0,C 180,E1 -26597.624,E2 -26597.624} C_VEL
LIN {X 0,Y 134.86,Z 384.305,A -85,B 0,C 180,E1 -26598.369,E2 -26598.369} C_VEL
LIN {X 0,Y 132.01,Z 376.52,A -85,B 0,C 180,E1 -26600.426,E2 -26600.426} C_VEL
LIN {X 0,Y 127.936,Z 368.962,A -85,B 0,C 180,E1 -26603.377,E2 -26603.377} C_VEL
LIN {X 0,Y 123.278,Z 361.452,A -85,B 0,C 180,E1 -26607.177,E2 -26607.177} C_VEL
LIN {X 0,Y 120.757,Z 357.7,A -85,B 0,C 180,E1 -26609.507,E2 -26609.507} C_VEL
LIN {X 0,Y 118.297,Z 354.134,A -85,B 0,C 180,E1 -26612.042,E2 -26612.042} C_VEL
LIN {X 0,Y 115.773,Z 350.732,A -85,B 0,C 180,E1 -26614.977,E2 -26614.977} C_VEL
LIN {X 0,Y 115.016,Z 349.663,A -85,B 0,C 180,E1 -26615.956,E2 -26615.956} C_VEL
LIN {X 0,Y 112.624,Z 347.158,A -85,B 0,C 180,E1 -26619.283,E2 -26619.283} C_VEL
LIN {X 0,Y 111.341,Z 344.626,A -85,B 0,C 180,E1 -26621.602,E2 -26621.602} C_VEL
LIN {X 0,Y 108.695,Z 342.605,A -85,B 0,C 180,E1 -26626.965,E2 -26626.965} C_VEL
LIN {X 0,Y 107.105,Z 339.334,A -85,B 0,C 180,E1 -26632.932,E2 -26632.932} C_VEL
LIN {X 0,Y 106.404,Z 338.375,A -85,B 0,C 180,E1 -26640,E2 -26640} C_VEL
LIN {X 0,Y 107.099,Z 339.3,A -85,B 0,C 180,E1 -26647.067,E2 -26647.067} C_VEL
LIN {X 0,Y 109.755,Z 343.723,A -85,B 0,C 180,E1 -26655.553,E2 -26655.553} C_VEL
LIN {X 0,Y 111.504,Z 344.974,A -85,B 0,C 180,E1 -26658.762,E2 -26658.762} C_VEL
LIN {X 0,Y 113.467,Z 348.29,A -85,B 0,C 180,E1 -26662.047,E2 -26662.047} C_VEL
LIN {X 0,Y 115.555,Z 350.289,A -85,B 0,C 180,E1 -26664.771,E2 -26664.771} C_VEL
LIN {X 0,Y 117.838,Z 353.662,A -85,B 0,C 180,E1 -26667.519,E2 -26667.519} C_VEL
LIN {X 0,Y 119.033,Z 355.148,A -85,B 0,C 180,E1 -26668.787,E2 -26668.787} C_VEL
LIN {X 0,Y 122.282,Z 359.959,A -85,B 0,C 180,E1 -26671.976,E2 -26671.976} C_VEL
LIN {X 0,Y 126.103,Z 365.851,A -85,B 0,C 180,E1 -26675.233,E2 -26675.233} C_VEL
LIN {X 0,Y 130.7,Z 373.927,A -85,B 0,C 180,E1 -26678.697,E2 -26678.697} C_VEL
LIN {X 0,Y 132.973,Z 378.88,A -85,B 0,C 180,E1 -26680.312,E2 -26680.312} C_VEL
LIN {X 0,Y 134.864,Z 384.295,A -85,B 0,C 180,E1 -26681.677,E2 -26681.677} C_VEL
LIN {X 0,Y 133.359,Z 402.334,A -85,B 0,C 180,E1 -26682.572,E2 -26682.572} C_VEL
LIN {X 0,Y 131.319,Z 414.114,A -85,B 0,C 180,E1 -26683.571,E2 -26683.571} C_VEL
LIN {X 0,Y 128.871,Z 423.813,A -85,B 0,C 180,E1 -26684.851,E2 -26684.851} C_VEL
LIN {X 0,Y 126.012,Z 432.774,A -85,B 0,C 180,E1 -26686.472,E2 -26686.472} C_VEL
LIN {X 0,Y 122.957,Z 440.725,A -85,B 0,C 180,E1 -26688.36,E2 -26688.36} C_VEL
LIN {X 0,Y 119.346,Z 448.552,A -85,B 0,C 180,E1 -26690.726,E2 -26690.726} C_VEL
LIN {X 0,Y 115.558,Z 455.872,A -85,B 0,C 180,E1 -26693.633,E2 -26693.633} C_VEL
LIN {X 0,Y 111.207,Z 463.295,A -85,B 0,C 180,E1 -26697.509,E2 -26697.509} C_VEL
LIN {X 0,Y 107.396,Z 469.108,A -85,B 0,C 180,E1 -26701.678,E2 -26701.678} C_VEL
LIN {X 0,Y 104.221,Z 473.692,A -85,B 0,C 180,E1 -26706.134,E2 -26706.134} C_VEL
LIN {X 0,Y 102.146,Z 476.671,A -85,B 0,C 180,E1 -26709.879,E2 -26709.879} C_VEL
LIN {X 0,Y 100.473,Z 478.983,A -85,B 0,C 180,E1 -26713.752,E2 -26713.752} C_VEL
LIN {X 0,Y 99.276,Z 480.711,A -85,B 0,C 180,E1 -26717.739,E2 -26717.739} C_VEL
LIN {X 0,Y 98.435,Z 481.947,A -85,B 0,C 180,E1 -26721.791,E2 -26721.791} C_VEL
LIN {X 0,Y 98.04,Z 482.712,A -85,B 0,C 180,E1 -26725.889,E2 -26725.889} C_VEL
LIN {X 0,Y 97.967,Z 483,A -85,B 0,C 180,E1 -26730,E2 -26730} C_VEL
LIN {X 0,Y 98.04,Z 482.699,A -85,B 0,C 180,E1 -26734.111,E2 -26734.111} C_VEL
LIN {X 0,Y 98.425,Z 481.909,A -85,B 0,C 180,E1 -26738.21,E2 -26738.21} C_VEL
LIN {X 0,Y 99.243,Z 480.647,A -85,B 0,C 180,E1 -26742.266,E2 -26742.266} C_VEL
LIN {X 0,Y 101.25,Z 477.741,A -85,B 0,C 180,E1 -26748.201,E2 -26748.201} C_VEL
LIN {X 0,Y 103.101,Z 475.09,A -85,B 0,C 180,E1 -26752.019,E2 -26752.019} C_VEL
LIN {X 0,Y 106.658,Z 469.912,A -85,B 0,C 180,E1 -26757.467,E2 -26757.467} C_VEL
LIN {X 0,Y 111.207,Z 463.076,A -85,B 0,C 180,E1 -26762.491,E2 -26762.491} C_VEL
LIN {X 0,Y 115.552,Z 455.607,A -85,B 0,C 180,E1 -26766.369,E2 -26766.369} C_VEL
LIN {X 0,Y 118.838,Z 449.259,A -85,B 0,C 180,E1 -26768.928,E2 -26768.928} C_VEL
LIN {X 0,Y 122.44,Z 441.572,A -85,B 0,C 180,E1 -26771.306,E2 -26771.306} C_VEL
LIN {X 0,Y 125.202,Z 434.538,A -85,B 0,C 180,E1 -26773.056,E2 -26773.056} C_VEL
LIN {X 0,Y 127.722,Z 426.975,A -85,B 0,C 180,E1 -26774.551,E2 -26774.551} C_VEL
LIN {X 0,Y 130.216,Z 417.869,A -85,B 0,C 180,E1 -26775.895,E2 -26775.895} C_VEL
LIN {X 0,Y 132.141,Z 408.614,A -85,B 0,C 180,E1 -26776.874,E2 -26776.874} C_VEL
LIN {X 0,Y 133.462,Z 399.633,A -85,B 0,C 180,E1 -26777.494,E2 -26777.494} C_VEL
LIN {X 0,Y 134.672,Z 384.063,A -85,B 0,C 180,E1 -26778.255,E2 -26778.255} C_VEL
LIN {X 0,Y 131.778,Z 376.243,A -85,B 0,C 180,E1 -26780.334,E2 -26780.334} C_VEL
LIN {X 0,Y 127.602,Z 368.519,A -85,B 0,C 180,E1 -26783.358,E2 -26783.358} C_VEL
LIN {X 0,Y 122.964,Z 361.079,A -85,B 0,C 180,E1 -26787.145,E2 -26787.145} C_VEL
LIN {X 0,Y 120.616,Z 357.597,A -85,B 0,C 180,E1 -26789.308,E2 -26789.308} C_VEL
LIN {X 0,Y 118.062,Z 353.921,A -85,B 0,C 180,E1 -26791.924,E2 -26791.924} C_VEL
LIN {X 0,Y 116.358,Z 351.808,A -85,B 0,C 180,E1 -26793.827,E2 -26793.827} C_VEL
LIN {X 0,Y 114.972,Z 350.381,A -85,B 0,C 180,E1 -26795.477,E2 -26795.477} C_VEL
LIN {X 0,Y 113.42,Z 350.09,A -85,B 0,C 180,E1 -26797.301,E2 -26797.301} C_VEL
LIN {X 0,Y 109.337,Z 351.023,A -85,B 0,C 180,E1 -26802.923,E2 -26802.923} C_VEL
LIN {X 0,Y 108.775,Z 350.804,A -85,B 0,C 180,E1 -26803.964,E2 -26803.964} C_VEL
LIN {X 0,Y 106.772,Z 348.328,A -85,B 0,C 180,E1 -26809.092,E2 -26809.092} C_VEL
LIN {X 0,Y 106.033,Z 346.233,A -85,B 0,C 180,E1 -26812.383,E2 -26812.383} C_VEL
LIN {X 0,Y 105.204,Z 345.317,A -85,B 0,C 180,E1 -26820,E2 -26820} C_VEL
LIN {X 0,Y 106.023,Z 346.224,A -85,B 0,C 180,E1 -26827.619,E2 -26827.619} C_VEL
LIN {X 0,Y 107.983,Z 350.144,A -85,B 0,C 180,E1 -26834.378,E2 -26834.378} C_VEL
LIN {X 0,Y 109.881,Z 351.735,A -85,B 0,C 180,E1 -26838.169,E2 -26838.169} C_VEL
LIN {X 0,Y 112.031,Z 355.237,A -85,B 0,C 180,E1 -26841.869,E2 -26841.869} C_VEL
LIN {X 0,Y 113.598,Z 356.95,A -85,B 0,C 180,E1 -26844.023,E2 -26844.023} C_VEL
LIN {X 0,Y 116.892,Z 361.721,A -85,B 0,C 180,E1 -26848.043,E2 -26848.043} C_VEL
LIN {X 0,Y 119.984,Z 366.517,A -85,B 0,C 180,E1 -26851.249,E2 -26851.249} C_VEL
LIN {X 0,Y 124.287,Z 373.753,A -85,B 0,C 180,E1 -26855.101,E2 -26855.101} C_VEL
LIN {X 0,Y 128.317,Z 381.607,A -85,B 0,C 180,E1 -26858.288,E2 -26858.288} C_VEL
LIN {X 0,Y 129.872,Z 386.249,A -85,B 0,C 180,E1 -26859.546,E2 -26859.546} C_VEL
LIN {X 0,Y 128.358,Z 402.961,A -85,B 0,C 180,E1 -26860.394,E2 -26860.394} C_VEL
LIN {X 0,Y 126.343,Z 414.021,A -85,B 0,C 180,E1 -26861.358,E2 -26861.358} C_VEL
LIN {X 0,Y 124.004,Z 423.08,A -85,B 0,C 180,E1 -26862.544,E2 -26862.544} C_VEL
LIN {X 0,Y 120.956,Z 432.323,A -85,B 0,C 180,E1 -26864.207,E2 -26864.207} C_VEL
LIN {X 0,Y 117.822,Z 440.245,A -85,B 0,C 180,E1 -26866.1,E2 -26866.1} C_VEL
LIN {X 0,Y 113.958,Z 448.157,A -85,B 0,C 180,E1 -26868.474,E2 -26868.474} C_VEL
LIN {X 0,Y 109.982,Z 455.539,A -85,B 0,C 180,E1 -26871.463,E2 -26871.463} C_VEL
LIN {X 0,Y 105.335,Z 463.02,A -85,B 0,C 180,E1 -26875.451,E2 -26875.451} C_VEL
LIN {X 0,Y 100.432,Z 469.873,A -85,B 0,C 180,E1 -26880.67,E2 -26880.67} C_VEL
LIN {X 0,Y 96.591,Z 475.059,A -85,B 0,C 180,E1 -26886.411,E2 -26886.411} C_VEL
LIN {X 0,Y 94.542,Z 477.718,A -85,B 0,C 180,E1 -26890.457,E2 -26890.457} C_VEL
LIN {X 0,Y 92.314,Z 480.631,A -85,B 0,C 180,E1 -26896.798,E2 -26896.798} C_VEL
LIN {X 0,Y 91.399,Z 481.899,A -85,B 0,C 180,E1 -26901.154,E2 -26901.154} C_VEL
LIN {X 0,Y 90.953,Z 482.696,A -85,B 0,C 180,E1 -26905.568,E2 -26905.568} C_VEL
LIN {X 0,Y 90.868,Z 482.999,A -85,B 0,C 180,E1 -26910,E2 -26910} C_VEL
LIN {X 0,Y 90.953,Z 482.715,A -85,B 0,C 180,E1 -26914.432,E2 -26914.432} C_VEL
LIN {X 0,Y 91.398,Z 481.957,A -85,B 0,C 180,E1 -26918.846,E2 -26918.846} C_VEL
LIN {X 0,Y 92.311,Z 480.728,A -85,B 0,C 180,E1 -26923.203,E2 -26923.203} C_VEL
LIN {X 0,Y 94.505,Z 477.855,A -85,B 0,C 180,E1 -26929.551,E2 -26929.551} C_VEL
LIN {X 0,Y 96.541,Z 475.24,A -85,B 0,C 180,E1 -26933.602,E2 -26933.602} C_VEL
LIN {X 0,Y 100.401,Z 470.102,A -85,B 0,C 180,E1 -26939.34,E2 -26939.34} C_VEL
LIN {X 0,Y 104.388,Z 464.576,A -85,B 0,C 180,E1 -26943.74,E2 -26943.74} C_VEL
LIN {X 0,Y 108.932,Z 457.628,A -85,B 0,C 180,E1 -26947.8,E2 -26947.8} C_VEL
LIN {X 0,Y 113.394,Z 449.653,A -85,B 0,C 180,E1 -26951.186,E2 -26951.186} C_VEL
LIN {X 0,Y 117.127,Z 442.229,A -85,B 0,C 180,E1 -26953.545,E2 -26953.545} C_VEL
LIN {X 0,Y 120.279,Z 434.647,A -85,B 0,C 180,E1 -26955.478,E2 -26955.478} C_VEL
LIN {X 0,Y 123.325,Z 426.019,A -85,B 0,C 180,E1 -26957.137,E2 -26957.137} C_VEL
LIN {X 0,Y 125.663,Z 417.455,A -85,B 0,C 180,E1 -26958.419,E2 -26958.419} C_VEL
LIN {X 0,Y 127.618,Z 408.629,A -85,B 0,C 180,E1 -26959.322,E2 -26959.322} C_VEL
LIN {X 0,Y 128.985,Z 399.075,A -85,B 0,C 180,E1 -26960.014,E2 -26960.014} C_VEL
LIN {X 0,Y 130.057,Z 386.331,A -85,B 0,C 180,E1 -26960.634,E2 -26960.634} C_VEL
LIN {X 0,Y 127.972,Z 380.673,A -85,B 0,C 180,E1 -26962.29,E2 -26962.29} C_VEL
LIN {X 0,Y 124.431,Z 373.857,A -85,B 0,C 180,E1 -26965.119,E2 -26965.119} C_VEL
LIN {X 0,Y 120.295,Z 366.89,A -85,B 0,C 180,E1 -26968.829,E2 -26968.829} C_VEL
LIN {X 0,Y 118.074,Z 363.456,A -85,B 0,C 180,E1 -26971.078,E2 -26971.078} C_VEL
LIN {X 0,Y 115.957,Z 360.254,A -85,B 0,C 180,E1 -26973.46,E2 -26973.46} C_VEL
LIN {X 0,Y 113.115,Z 356.159,A -85,B 0,C 180,E1 -26977.149,E2 -26977.149} C_VEL
LIN {X 0,Y 110.612,Z 353.106,A -85,B 0,C 180,E1 -26981.038,E2 -26981.038} C_VEL
LIN {X 0,Y 109.745,Z 351.378,A -85,B 0,C 180,E1 -26982.771,E2 -26982.771} C_VEL
LIN {X 0,Y 107.358,Z 349.234,A -85,B 0,C 180,E1 -26988.173,E2 -26988.173} C_VEL
LIN {X 0,Y 106.089,Z 346.24,A -85,B 0,C 180,E1 -26993.674,E2 -26993.674} C_VEL
LIN {X 0,Y 105.537,Z 345.434,A -85,B 0,C 180,E1 -27000,E2 -27000} C_VEL
LIN {X 0,Y 106.172,Z 346.368,A -85,B 0,C 180,E1 -27006.835,E2 -27006.835} C_VEL
LIN {X 0,Y 108.324,Z 350.413,A -85,B 0,C 180,E1 -27014.412,E2 -27014.412} C_VEL
LIN {X 0,Y 109.943,Z 351.721,A -85,B 0,C 180,E1 -27017.676,E2 -27017.676} C_VEL
LIN {X 0,Y 112.041,Z 355.146,A -85,B 0,C 180,E1 -27021.383,E2 -27021.383} C_VEL
LIN {X 0,Y 113.614,Z 356.812,A -85,B 0,C 180,E1 -27023.587,E2 -27023.587} C_VEL
LIN {X 0,Y 116.2,Z 360.505,A -85,B 0,C 180,E1 -27026.858,E2 -27026.858} C_VEL
LIN {X 0,Y 119.822,Z 366.153,A -85,B 0,C 180,E1 -27030.756,E2 -27030.756} C_VEL
LIN {X 0,Y 123.053,Z 371.397,A -85,B 0,C 180,E1 -27033.743,E2 -27033.743} C_VEL
LIN {X 0,Y 127.333,Z 379.312,A -85,B 0,C 180,E1 -27037.258,E2 -27037.258} C_VEL
LIN {X 0,Y 129.331,Z 384.145,A -85,B 0,C 180,E1 -27038.828,E2 -27038.828} C_VEL
LIN {X 0,Y 130.084,Z 386.408,A -85,B 0,C 180,E1 -27039.432,E2 -27039.432} C_VEL
LIN {X 0,Y 128.556,Z 403.398,A -85,B 0,C 180,E1 -27040.312,E2 -27040.312} C_VEL
LIN {X 0,Y 126.531,Z 414.102,A -85,B 0,C 180,E1 -27041.237,E2 -27041.237} C_VEL
LIN {X 0,Y 123.964,Z 423.819,A -85,B 0,C 180,E1 -27042.523,E2 -27042.523} C_VEL
LIN {X 0,Y 121.079,Z 432.47,A -85,B 0,C 180,E1 -27044.089,E2 -27044.089} C_VEL
LIN {X 0,Y 117.747,Z 440.729,A -85,B 0,C 180,E1 -27046.064,E2 -27046.064} C_VEL
LIN {X 0,Y 113.952,Z 448.555,A -85,B 0,C 180,E1 -27048.472,E2 -27048.472} C_VEL
LIN {X 0,Y 109.924,Z 455.874,A -85,B 0,C 180,E1 -27051.439,E2 -27051.439} C_VEL
LIN {X 0,Y 105.291,Z 463.297,A -85,B 0,C 180,E1 -27055.434,E2 -27055.434} C_VEL
LIN {X 0,Y 101.208,Z 469.109,A -85,B 0,C 180,E1 -27059.772,E2 -27059.772} C_VEL
LIN {X 0,Y 97.749,Z 473.693,A -85,B 0,C 180,E1 -27064.445,E2 -27064.445} C_VEL
LIN {X 0,Y 95.488,Z 476.672,A -85,B 0,C 180,E1 -27068.408,E2 -27068.408} C_VEL
LIN {X 0,Y 93.676,Z 478.983,A -85,B 0,C 180,E1 -27072.537,E2 -27072.537} C_VEL
LIN {X 0,Y 92.337,Z 480.712,A -85,B 0,C 180,E1 -27076.801,E2 -27076.801} C_VEL
LIN {X 0,Y 91.406,Z 481.947,A -85,B 0,C 180,E1 -27081.154,E2 -27081.154} C_VEL
LIN {X 0,Y 90.952,Z 482.712,A -85,B 0,C 180,E1 -27085.568,E2 -27085.568} C_VEL
LIN {X 0,Y 90.866,Z 483,A -85,B 0,C 180,E1 -27090,E2 -27090} C_VEL
LIN {X 0,Y 90.951,Z 482.699,A -85,B 0,C 180,E1 -27094.432,E2 -27094.432} C_VEL
LIN {X 0,Y 91.397,Z 481.908,A -85,B 0,C 180,E1 -27098.846,E2 -27098.846} C_VEL
LIN {X 0,Y 92.31,Z 480.647,A -85,B 0,C 180,E1 -27103.203,E2 -27103.203} C_VEL
LIN {X 0,Y 94.513,Z 477.741,A -85,B 0,C 180,E1 -27109.549,E2 -27109.549} C_VEL
LIN {X 0,Y 96.547,Z 475.089,A -85,B 0,C 180,E1 -27113.6,E2 -27113.6} C_VEL
LIN {X 0,Y 100.405,Z 469.91,A -85,B 0,C 180,E1 -27119.338,E2 -27119.338} C_VEL
LIN {X 0,Y 105.292,Z 463.073,A -85,B 0,C 180,E1 -27124.565,E2 -27124.565} C_VEL
LIN {X 0,Y 109.922,Z 455.605,A -85,B 0,C 180,E1 -27128.562,E2 -27128.562} C_VEL
LIN {X 0,Y 113.945,Z 448.235,A -85,B 0,C 180,E1 -27131.531,E2 -27131.531} C_VEL
LIN {X 0,Y 117.698,Z 440.478,A -85,B 0,C 180,E1 -27133.891,E2 -27133.891} C_VEL
LIN {X 0,Y 120.999,Z 432.138,A -85,B 0,C 180,E1 -27135.891,E2 -27135.891} C_VEL
LIN {X 0,Y 124.275,Z 422.176,A -85,B 0,C 180,E1 -27137.654,E2 -27137.654} C_VEL
LIN {X 0,Y 127.129,Z 410.267,A -85,B 0,C 180,E1 -27139.04,E2 -27139.04} C_VEL
LIN {X 0,Y 128.649,Z 400.817,A -85,B 0,C 180,E1 -27139.748,E2 -27139.748} C_VEL
LIN {X 0,Y 129.911,Z 386.35,A -85,B 0,C 180,E1 -27140.469,E2 -27140.469} C_VEL
LIN {X 0,Y 127.795,Z 380.493,A -85,B 0,C 180,E1 -27142.155,E2 -27142.155} C_VEL
LIN {X 0,Y 124.22,Z 373.68,A -85,B 0,C 180,E1 -27144.996,E2 -27144.996} C_VEL
LIN {X 0,Y 120.194,Z 366.811,A -85,B 0,C 180,E1 -27148.598,E2 -27148.598} C_VEL
LIN {X 0,Y 116.117,Z 360.453,A -85,B 0,C 180,E1 -27152.897,E2 -27152.897} C_VEL
LIN {X 0,Y 113.482,Z 356.734,A -85,B 0,C 180,E1 -27156.186,E2 -27156.186} C_VEL
LIN {X 0,Y 110.349,Z 352.752,A -85,B 0,C 180,E1 -27160.95,E2 -27160.95} C_VEL
LIN {X 0,Y 109.68,Z 351.347,A -85,B 0,C 180,E1 -27162.28,E2 -27162.28} C_VEL
LIN {X 0,Y 108.775,Z 350.804,A -85,B 0,C 180,E1 -27163.964,E2 -27163.964} C_VEL
LIN {X 0,Y 106.928,Z 350.213,A -85,B 0,C 180,E1 -27168.054,E2 -27168.054} C_VEL
LIN {X 0,Y 104.984,Z 351.185,A -85,B 0,C 180,E1 -27174.429,E2 -27174.429} C_VEL
LIN {X 0,Y 104.344,Z 352.444,A -85,B 0,C 180,E1 -27180.983,E2 -27180.983} C_VEL
LIN {X 0,Y 105.05,Z 353.289,A -85,B 0,C 180,E1 -27187.207,E2 -27187.207} C_VEL
LIN {X 0,Y 106.633,Z 356.831,A -85,B 0,C 180,E1 -27193.282,E2 -27193.282} C_VEL
LIN {X 0,Y 108.362,Z 358.467,A -85,B 0,C 180,E1 -27197.091,E2 -27197.091} C_VEL
LIN {X 0,Y 110.673,Z 362.189,A -85,B 0,C 180,E1 -27201.295,E2 -27201.295} C_VEL
LIN {X 0,Y 111.846,Z 363.703,A -85,B 0,C 180,E1 -27203.033,E2 -27203.033} C_VEL
LIN {X 0,Y 114.669,Z 367.987,A -85,B 0,C 180,E1 -27206.746,E2 -27206.746} C_VEL
LIN {X 0,Y 118.139,Z 373.563,A -85,B 0,C 180,E1 -27210.576,E2 -27210.576} C_VEL
LIN {X 0,Y 122.756,Z 382.212,A -85,B 0,C 180,E1 -27214.926,E2 -27214.926} C_VEL
LIN {X 0,Y 124.948,Z 387.34,A -85,B 0,C 180,E1 -27216.827,E2 -27216.827} C_VEL
LIN {X 0,Y 125.287,Z 388.471,A -85,B 0,C 180,E1 -27217.139,E2 -27217.139} C_VEL
LIN {X 0,Y 123.757,Z 403.857,A -85,B 0,C 180,E1 -27217.946,E2 -27217.946} C_VEL
LIN {X 0,Y 121.496,Z 415.1,A -85,B 0,C 180,E1 -27218.982,E2 -27218.982} C_VEL
LIN {X 0,Y 119.335,Z 423.086,A -85,B 0,C 180,E1 -27220.04,E2 -27220.04} C_VEL
LIN {X 0,Y 116.288,Z 431.909,A -85,B 0,C 180,E1 -27221.608,E2 -27221.608} C_VEL
LIN {X 0,Y 112.824,Z 440.249,A -85,B 0,C 180,E1 -27223.604,E2 -27223.604} C_VEL
LIN {X 0,Y 108.756,Z 448.161,A -85,B 0,C 180,E1 -27226,E2 -27226} C_VEL
LIN {X 0,Y 104.522,Z 455.542,A -85,B 0,C 180,E1 -27229.037,E2 -27229.037} C_VEL
LIN {X 0,Y 99.572,Z 463.022,A -85,B 0,C 180,E1 -27233.135,E2 -27233.135} C_VEL
LIN {X 0,Y 94.303,Z 469.874,A -85,B 0,C 180,E1 -27238.556,E2 -27238.556} C_VEL
LIN {X 0,Y 90.119,Z 475.06,A -85,B 0,C 180,E1 -27244.601,E2 -27244.601} C_VEL
LIN {X 0,Y 87.871,Z 477.719,A -85,B 0,C 180,E1 -27248.906,E2 -27248.906} C_VEL
LIN {X 0,Y 85.422,Z 480.631,A -85,B 0,C 180,E1 -27255.711,E2 -27255.711} C_VEL
LIN {X 0,Y 84.398,Z 481.899,A -85,B 0,C 180,E1 -27260.413,E2 -27260.413} C_VEL
LIN {X 0,Y 83.888,Z 482.696,A -85,B 0,C 180,E1 -27265.194,E2 -27265.194} C_VEL
LIN {X 0,Y 83.784,Z 482.999,A -85,B 0,C 180,E1 -27270,E2 -27270} C_VEL
LIN {X 0,Y 83.888,Z 482.715,A -85,B 0,C 180,E1 -27274.806,E2 -27274.806} C_VEL
LIN {X 0,Y 84.397,Z 481.956,A -85,B 0,C 180,E1 -27279.587,E2 -27279.587} C_VEL
LIN {X 0,Y 85.418,Z 480.727,A -85,B 0,C 180,E1 -27284.29,E2 -27284.29} C_VEL
LIN {X 0,Y 87.834,Z 477.854,A -85,B 0,C 180,E1 -27291.104,E2 -27291.104} C_VEL
LIN {X 0,Y 90.076,Z 475.239,A -85,B 0,C 180,E1 -27295.411,E2 -27295.411} C_VEL
LIN {X 0,Y 94.273,Z 470.101,A -85,B 0,C 180,E1 -27301.455,E2 -27301.455} C_VEL
LIN {X 0,Y 98.554,Z 464.575,A -85,B 0,C 180,E1 -27306.037,E2 -27306.037} C_VEL
LIN {X 0,Y 103.422,Z 457.625,A -85,B 0,C 180,E1 -27310.207,E2 -27310.207} C_VEL
LIN {X 0,Y 108.162,Z 449.65,A -85,B 0,C 180,E1 -27313.658,E2 -27313.658} C_VEL
LIN {X 0,Y 111.918,Z 442.604,A -85,B 0,C 180,E1 -27315.937,E2 -27315.937} C_VEL
LIN {X 0,Y 115.645,Z 434.078,A -85,B 0,C 180,E1 -27318.108,E2 -27318.108} C_VEL
LIN {X 0,Y 118.655,Z 425.828,A -85,B 0,C 180,E1 -27319.691,E2 -27319.691} C_VEL
LIN {X 0,Y 121.248,Z 416.771,A -85,B 0,C 180,E1 -27321.012,E2 -27321.012} C_VEL
LIN {X 0,Y 123.469,Z 406.736,A -85,B 0,C 180,E1 -27321.99,E2 -27321.99} C_VEL
LIN {X 0,Y 125.033,Z 394.939,A -85,B 0,C 180,E1 -27322.721,E2 -27322.721} C_VEL
LIN {X 0,Y 125.483,Z 388.406,A -85,B 0,C 180,E1 -27323.058,E2 -27323.058} C_VEL
LIN {X 0,Y 123.355,Z 383.3,A -85,B 0,C 180,E1 -27324.894,E2 -27324.894} C_VEL
LIN {X 0,Y 119.593,Z 376.052,A -85,B 0,C 180,E1 -27328.347,E2 -27328.347} C_VEL
LIN {X 0,Y 115.768,Z 369.612,A -85,B 0,C 180,E1 -27332.395,E2 -27332.395} C_VEL
LIN {X 0,Y 113.53,Z 366.119,A -85,B 0,C 180,E1 -27335.148,E2 -27335.148} C_VEL
LIN {X 0,Y 111.166,Z 362.536,A -85,B 0,C 180,E1 -27338.531,E2 -27338.531} C_VEL
LIN {X 0,Y 108.785,Z 359.19,A -85,B 0,C 180,E1 -27342.696,E2 -27342.696} C_VEL
LIN {X 0,Y 108.173,Z 358.081,A -85,B 0,C 180,E1 -27344.025,E2 -27344.025} C_VEL
LIN {X 0,Y 106.05,Z 355.784,A -85,B 0,C 180,E1 -27349.499,E2 -27349.499} C_VEL
LIN {X 0,Y 105.118,Z 353.198,A -85,B 0,C 180,E1 -27354.244,E2 -27354.244} C_VEL
LIN {X 0,Y 104.671,Z 352.49,A -85,B 0,C 180,E1 -27360,E2 -27360} C_VEL
LIN {X 0,Y 105.194,Z 353.408,A -85,B 0,C 180,E1 -27366.325,E2 -27366.325} C_VEL
LIN {X 0,Y 106.959,Z 357.123,A -85,B 0,C 180,E1 -27373.295,E2 -27373.295} C_VEL
LIN {X 0,Y 108.494,Z 358.541,A -85,B 0,C 180,E1 -27376.705,E2 -27376.705} C_VEL
LIN {X 0,Y 110.625,Z 362.002,A -85,B 0,C 180,E1 -27380.694,E2 -27380.694} C_VEL
LIN {X 0,Y 111.701,Z 363.231,A -85,B 0,C 180,E1 -27382.316,E2 -27382.316} C_VEL
LIN {X 0,Y 114.799,Z 368.089,A -85,B 0,C 180,E1 -27386.502,E2 -27386.502} C_VEL
LIN {X 0,Y 118.335,Z 373.748,A -85,B 0,C 180,E1 -27390.427,E2 -27390.427} C_VEL
LIN {X 0,Y 123.007,Z 382.539,A -85,B 0,C 180,E1 -27394.844,E2 -27394.844} C_VEL
LIN {X 0,Y 125.05,Z 387.222,A -85,B 0,C 180,E1 -27396.612,E2 -27396.612} C_VEL
LIN {X 0,Y 125.51,Z 388.688,A -85,B 0,C 180,E1 -27397.03,E2 -27397.03} C_VEL
LIN {X 0,Y 123.961,Z 404.252,A -85,B 0,C 180,E1 -27397.869,E2 -27397.869} C_VEL
LIN {X 0,Y 121.7,Z 415.211,A -85,B 0,C 180,E1 -27398.871,E2 -27398.871} C_VEL
LIN {X 0,Y 119.292,Z 423.825,A -85,B 0,C 180,E1 -27400.016,E2 -27400.016} C_VEL
LIN {X 0,Y 116.256,Z 432.475,A -85,B 0,C 180,E1 -27401.578,E2 -27401.578} C_VEL
LIN {X 0,Y 112.816,Z 440.573,A -85,B 0,C 180,E1 -27403.516,E2 -27403.516} C_VEL
LIN {X 0,Y 109.318,Z 447.538,A -85,B 0,C 180,E1 -27405.643,E2 -27405.643} C_VEL
LIN {X 0,Y 105.476,Z 454.173,A -85,B 0,C 180,E1 -27408.218,E2 -27408.218} C_VEL
LIN {X 0,Y 101.441,Z 460.473,A -85,B 0,C 180,E1 -27411.427,E2 -27411.427} C_VEL
LIN {X 0,Y 97.677,Z 465.705,A -85,B 0,C 180,E1 -27414.858,E2 -27414.858} C_VEL
LIN {X 0,Y 94.284,Z 470.067,A -85,B 0,C 180,E1 -27418.549,E2 -27418.549} C_VEL
LIN {X 0,Y 90.087,Z 475.211,A -85,B 0,C 180,E1 -27424.592,E2 -27424.592} C_VEL
LIN {X 0,Y 86.933,Z 478.984,A -85,B 0,C 180,E1 -27431.133,E2 -27431.133} C_VEL
LIN {X 0,Y 85.439,Z 480.712,A -85,B 0,C 180,E1 -27435.714,E2 -27435.714} C_VEL
LIN {X 0,Y 84.404,Z 481.947,A -85,B 0,C 180,E1 -27440.414,E2 -27440.414} C_VEL
LIN {X 0,Y 83.887,Z 482.712,A -85,B 0,C 180,E1 -27445.194,E2 -27445.194} C_VEL
LIN {X 0,Y 83.782,Z 483,A -85,B 0,C 180,E1 -27450,E2 -27450} C_VEL
LIN {X 0,Y 83.886,Z 482.699,A -85,B 0,C 180,E1 -27454.806,E2 -27454.806} C_VEL
LIN {X 0,Y 84.396,Z 481.908,A -85,B 0,C 180,E1 -27459.587,E2 -27459.587} C_VEL
LIN {X 0,Y 85.417,Z 480.646,A -85,B 0,C 180,E1 -27464.29,E2 -27464.29} C_VEL
LIN {X 0,Y 87.843,Z 477.74,A -85,B 0,C 180,E1 -27471.101,E2 -27471.101} C_VEL
LIN {X 0,Y 90.081,Z 475.088,A -85,B 0,C 180,E1 -27475.41,E2 -27475.41} C_VEL
LIN {X 0,Y 94.279,Z 469.909,A -85,B 0,C 180,E1 -27481.453,E2 -27481.453} C_VEL
LIN {X 0,Y 99.519,Z 463.071,A -85,B 0,C 180,E1 -27486.888,E2 -27486.888} C_VEL
LIN {X 0,Y 104.458,Z 455.602,A -85,B 0,C 180,E1 -27490.993,E2 -27490.993} C_VEL
LIN {X 0,Y 108.739,Z 448.232,A -85,B 0,C 180,E1 -27494.009,E2 -27494.009} C_VEL
LIN {X 0,Y 112.755,Z 440.333,A -85,B 0,C 180,E1 -27496.433,E2 -27496.433} C_VEL
LIN {X 0,Y 116.827,Z 430.484,A -85,B 0,C 180,E1 -27498.757,E2 -27498.757} C_VEL
LIN {X 0,Y 120.518,Z 418.895,A -85,B 0,C 180,E1 -27500.598,E2 -27500.598} C_VEL
LIN {X 0,Y 122.706,Z 409.508,A -85,B 0,C 180,E1 -27501.628,E2 -27501.628} C_VEL
LIN {X 0,Y 124.178,Z 400.801,A -85,B 0,C 180,E1 -27502.25,E2 -27502.25} C_VEL
LIN {X 0,Y 125.366,Z 388.641,A -85,B 0,C 180,E1 -27502.842,E2 -27502.842} C_VEL
LIN {X 0,Y 123.845,Z 384.492,A -85,B 0,C 180,E1 -27504.181,E2 -27504.181} C_VEL
LIN {X 0,Y 119.659,Z 376.333,A -85,B 0,C 180,E1 -27507.95,E2 -27507.95} C_VEL
LIN {X 0,Y 115.827,Z 369.777,A -85,B 0,C 180,E1 -27511.95,E2 -27511.95} C_VEL
LIN {X 0,Y 113.408,Z 366.067,A -85,B 0,C 180,E1 -27514.872,E2 -27514.872} C_VEL
LIN {X 0,Y 111.072,Z 362.484,A -85,B 0,C 180,E1 -27518.178,E2 -27518.178} C_VEL
LIN {X 0,Y 108.692,Z 359.223,A -85,B 0,C 180,E1 -27522.236,E2 -27522.236} C_VEL
LIN {X 0,Y 108.114,Z 358.077,A -85,B 0,C 180,E1 -27523.477,E2 -27523.477} C_VEL
LIN {X 0,Y 105.882,Z 355.708,A -85,B 0,C 180,E1 -27528.999,E2 -27528.999} C_VEL
LIN {X 0,Y 104.973,Z 353.126,A -85,B 0,C 180,E1 -27533.272,E2 -27533.272} C_VEL
LIN {X 0,Y 104.344,Z 352.444,A -85,B 0,C 180,E1 -27540.983,E2 -27540.983} C_VEL
LIN {X 0,Y 104.47,Z 353.504,A -85,B 0,C 180,E1 -27544.154,E2 -27544.154} C_VEL
LIN {X 0,Y 104.745,Z 355.674,A -85,B 0,C 180,E1 -27547.164,E2 -27547.164} C_VEL
LIN {X 0,Y 107.11,Z 365.732,A -85,B 0,C 180,E1 -27556.526,E2 -27556.526} C_VEL
LIN {X 0,Y 109.95,Z 370.1,A -85,B 0,C 180,E1 -27561.718,E2 -27561.718} C_VEL
LIN {X 0,Y 112.485,Z 374.181,A -85,B 0,C 180,E1 -27565.365,E2 -27565.365} C_VEL
LIN {X 0,Y 115.637,Z 379.665,A -85,B 0,C 180,E1 -27569.177,E2 -27569.177} C_VEL
LIN {X 0,Y 119.619,Z 387.64,A -85,B 0,C 180,E1 -27573.297,E2 -27573.297} C_VEL
LIN {X 0,Y 120.937,Z 390.605,A -85,B 0,C 180,E1 -27574.543,E2 -27574.543} C_VEL
LIN {X 0,Y 119.33,Z 405.042,A -85,B 0,C 180,E1 -27575.355,E2 -27575.355} C_VEL
LIN {X 0,Y 116.865,Z 416.215,A -85,B 0,C 180,E1 -27576.419,E2 -27576.419} C_VEL
LIN {X 0,Y 114.254,Z 424.966,A -85,B 0,C 180,E1 -27577.632,E2 -27577.632} C_VEL
LIN {X 0,Y 110.973,Z 433.683,A -85,B 0,C 180,E1 -27579.269,E2 -27579.269} C_VEL
LIN {X 0,Y 107.24,Z 441.885,A -85,B 0,C 180,E1 -27581.327,E2 -27581.327} C_VEL
LIN {X 0,Y 102.616,Z 450.206,A -85,B 0,C 180,E1 -27584.019,E2 -27584.019} C_VEL
LIN {X 0,Y 97.108,Z 458.775,A -85,B 0,C 180,E1 -27587.977,E2 -27587.977} C_VEL
LIN {X 0,Y 91.981,Z 465.469,A -85,B 0,C 180,E1 -27592.321,E2 -27592.321} C_VEL
LIN {X 0,Y 88.324,Z 469.876,A -85,B 0,C 180,E1 -27596.153,E2 -27596.153} C_VEL
LIN {X 0,Y 83.754,Z 475.062,A -85,B 0,C 180,E1 -27602.516,E2 -27602.516} C_VEL
LIN {X 0,Y 81.281,Z 477.719,A -85,B 0,C 180,E1 -27607.102,E2 -27607.102} C_VEL
LIN {X 0,Y 78.551,Z 480.632,A -85,B 0,C 180,E1 -27614.431,E2 -27614.431} C_VEL
LIN {X 0,Y 77.403,Z 481.899,A -85,B 0,C 180,E1 -27619.538,E2 -27619.538} C_VEL
LIN {X 0,Y 76.812,Z 482.696,A -85,B 0,C 180,E1 -27624.75,E2 -27624.75} C_VEL
LIN {X 0,Y 76.693,Z 482.999,A -85,B 0,C 180,E1 -27630,E2 -27630} C_VEL
LIN {X 0,Y 76.812,Z 482.715,A -85,B 0,C 180,E1 -27635.25,E2 -27635.25} C_VEL
LIN {X 0,Y 77.403,Z 481.956,A -85,B 0,C 180,E1 -27640.462,E2 -27640.462} C_VEL
LIN {X 0,Y 78.547,Z 480.727,A -85,B 0,C 180,E1 -27645.57,E2 -27645.57} C_VEL
LIN {X 0,Y 81.245,Z 477.853,A -85,B 0,C 180,E1 -27652.908,E2 -27652.908} C_VEL
LIN {X 0,Y 83.718,Z 475.237,A -85,B 0,C 180,E1 -27657.497,E2 -27657.497} C_VEL
LIN {X 0,Y 88.295,Z 470.099,A -85,B 0,C 180,E1 -27663.86,E2 -27663.86} C_VEL
LIN {X 0,Y 92.901,Z 464.573,A -85,B 0,C 180,E1 -27668.616,E2 -27668.616} C_VEL
LIN {X 0,Y 98.11,Z 457.623,A -85,B 0,C 180,E1 -27672.883,E2 -27672.883} C_VEL
LIN {X 0,Y 103.155,Z 449.647,A -85,B 0,C 180,E1 -27676.375,E2 -27676.375} C_VEL
LIN {X 0,Y 106.91,Z 443.008,A -85,B 0,C 180,E1 -27678.548,E2 -27678.548} C_VEL
LIN {X 0,Y 111.036,Z 434.074,A -85,B 0,C 180,E1 -27680.833,E2 -27680.833} C_VEL
LIN {X 0,Y 114.199,Z 425.822,A -85,B 0,C 180,E1 -27682.403,E2 -27682.403} C_VEL
LIN {X 0,Y 116.7,Z 417.603,A -85,B 0,C 180,E1 -27683.607,E2 -27683.607} C_VEL
LIN {X 0,Y 118.958,Z 408.049,A -85,B 0,C 180,E1 -27684.571,E2 -27684.571} C_VEL
LIN {X 0,Y 120.472,Z 398.303,A -85,B 0,C 180,E1 -27685.224,E2 -27685.224} C_VEL
LIN {X 0,Y 121.077,Z 390.661,A -85,B 0,C 180,E1 -27685.691,E2 -27685.691} C_VEL
LIN {X 0,Y 118.194,Z 384.471,A -85,B 0,C 180,E1 -27688.492,E2 -27688.492} C_VEL
LIN {X 0,Y 114.744,Z 377.927,A -85,B 0,C 180,E1 -27692.273,E2 -27692.273} C_VEL
LIN {X 0,Y 111.766,Z 372.762,A -85,B 0,C 180,E1 -27696.121,E2 -27696.121} C_VEL
LIN {X 0,Y 109.386,Z 369.019,A -85,B 0,C 180,E1 -27699.797,E2 -27699.797} C_VEL
LIN {X 0,Y 107.041,Z 365.276,A -85,B 0,C 180,E1 -27704.428,E2 -27704.428} C_VEL
LIN {X 0,Y 104.509,Z 361.589,A -85,B 0,C 180,E1 -27712.27,E2 -27712.27} C_VEL
LIN {X 0,Y 104.114,Z 360.077,A -85,B 0,C 180,E1 -27715.159,E2 -27715.159} C_VEL
LIN {X 0,Y 103.804,Z 359.546,A -85,B 0,C 180,E1 -27720,E2 -27720} C_VEL
LIN {X 0,Y 104.187,Z 360.259,A -85,B 0,C 180,E1 -27725.467,E2 -27725.467} C_VEL
LIN {X 0,Y 105.921,Z 364.139,A -85,B 0,C 180,E1 -27732.94,E2 -27732.94} C_VEL
LIN {X 0,Y 107.052,Z 365.269,A -85,B 0,C 180,E1 -27735.636,E2 -27735.636} C_VEL
LIN {X 0,Y 109.16,Z 368.779,A -85,B 0,C 180,E1 -27739.878,E2 -27739.878} C_VEL
LIN {X 0,Y 110.151,Z 370.279,A -85,B 0,C 180,E1 -27741.522,E2 -27741.522} C_VEL
LIN {X 0,Y 112.576,Z 374.163,A -85,B 0,C 180,E1 -27745.045,E2 -27745.045} C_VEL
LIN {X 0,Y 115.844,Z 379.882,A -85,B 0,C 180,E1 -27749.035,E2 -27749.035} C_VEL
LIN {X 0,Y 119.782,Z 387.713,A -85,B 0,C 180,E1 -27753.121,E2 -27753.121} C_VEL
LIN {X 0,Y 121.234,Z 391.097,A -85,B 0,C 180,E1 -27754.507,E2 -27754.507} C_VEL
LIN {X 0,Y 119.453,Z 405.677,A -85,B 0,C 180,E1 -27755.289,E2 -27755.289} C_VEL
LIN {X 0,Y 117.08,Z 416.323,A -85,B 0,C 180,E1 -27756.308,E2 -27756.308} C_VEL
LIN {X 0,Y 114.509,Z 424.861,A -85,B 0,C 180,E1 -27757.474,E2 -27757.474} C_VEL
LIN {X 0,Y 111.427,Z 433.058,A -85,B 0,C 180,E1 -27758.974,E2 -27758.974} C_VEL
LIN {X 0,Y 107.697,Z 441.293,A -85,B 0,C 180,E1 -27760.983,E2 -27760.983} C_VEL
LIN {X 0,Y 103.773,Z 448.561,A -85,B 0,C 180,E1 -27763.279,E2 -27763.279} C_VEL
LIN {X 0,Y 99.21,Z 455.88,A -85,B 0,C 180,E1 -27766.317,E2 -27766.317} C_VEL
LIN {X 0,Y 93.923,Z 463.301,A -85,B 0,C 180,E1 -27770.505,E2 -27770.505} C_VEL
LIN {X 0,Y 89.197,Z 469.112,A -85,B 0,C 180,E1 -27775.164,E2 -27775.164} C_VEL
LIN {X 0,Y 85.123,Z 473.695,A -85,B 0,C 180,E1 -27780.306,E2 -27780.306} C_VEL
LIN {X 0,Y 82.426,Z 476.674,A -85,B 0,C 180,E1 -27784.766,E2 -27784.766} C_VEL
LIN {X 0,Y 80.228,Z 478.985,A -85,B 0,C 180,E1 -27789.489,E2 -27789.489} C_VEL
LIN {X 0,Y 78.564,Z 480.713,A -85,B 0,C 180,E1 -27794.433,E2 -27794.433} C_VEL
LIN {X 0,Y 77.409,Z 481.948,A -85,B 0,C 180,E1 -27799.538,E2 -27799.538} C_VEL
LIN {X 0,Y 76.812,Z 482.712,A -85,B 0,C 180,E1 -27804.75,E2 -27804.75} C_VEL
LIN {X 0,Y 76.692,Z 483,A -85,B 0,C 180,E1 -27810,E2 -27810} C_VEL
LIN {X 0,Y 76.811,Z 482.699,A -85,B 0,C 180,E1 -27815.25,E2 -27815.25} C_VEL
LIN {X 0,Y 77.401,Z 481.908,A -85,B 0,C 180,E1 -27820.463,E2 -27820.463} C_VEL
LIN {X 0,Y 78.546,Z 480.646,A -85,B 0,C 180,E1 -27825.57,E2 -27825.57} C_VEL
LIN {X 0,Y 81.254,Z 477.739,A -85,B 0,C 180,E1 -27832.906,E2 -27832.906} C_VEL
LIN {X 0,Y 83.721,Z 475.087,A -85,B 0,C 180,E1 -27837.496,E2 -27837.496} C_VEL
LIN {X 0,Y 88.302,Z 469.907,A -85,B 0,C 180,E1 -27843.857,E2 -27843.857} C_VEL
LIN {X 0,Y 93.925,Z 463.069,A -85,B 0,C 180,E1 -27849.494,E2 -27849.494} C_VEL
LIN {X 0,Y 99.196,Z 455.599,A -85,B 0,C 180,E1 -27853.691,E2 -27853.691} C_VEL
LIN {X 0,Y 103.759,Z 448.229,A -85,B 0,C 180,E1 -27856.729,E2 -27856.729} C_VEL
LIN {X 0,Y 107.631,Z 441.038,A -85,B 0,C 180,E1 -27858.97,E2 -27858.97} C_VEL
LIN {X 0,Y 110.913,Z 433.778,A -85,B 0,C 180,E1 -27860.769,E2 -27860.769} C_VEL
LIN {X 0,Y 114.17,Z 425.083,A -85,B 0,C 180,E1 -27862.422,E2 -27862.422} C_VEL
LIN {X 0,Y 116.865,Z 416.253,A -85,B 0,C 180,E1 -27863.615,E2 -27863.615} C_VEL
LIN {X 0,Y 119.34,Z 405.054,A -85,B 0,C 180,E1 -27864.681,E2 -27864.681} C_VEL
LIN {X 0,Y 120.964,Z 391.638,A -85,B 0,C 180,E1 -27865.378,E2 -27865.378} C_VEL
LIN {X 0,Y 120.777,Z 390.231,A -85,B 0,C 180,E1 -27865.652,E2 -27865.652} C_VEL
LIN {X 0,Y 117.46,Z 383.214,A -85,B 0,C 180,E1 -27868.898,E2 -27868.898} C_VEL
LIN {X 0,Y 113.724,Z 376.168,A -85,B 0,C 180,E1 -27873.119,E2 -27873.119} C_VEL
LIN {X 0,Y 111.223,Z 372.154,A -85,B 0,C 180,E1 -27876.407,E2 -27876.407} C_VEL
LIN {X 0,Y 109.187,Z 368.905,A -85,B 0,C 180,E1 -27879.575,E2 -27879.575} C_VEL
LIN {X 0,Y 106.883,Z 365.192,A -85,B 0,C 180,E1 -27884.064,E2 -27884.064} C_VEL
LIN {X 0,Y 104.425,Z 361.801,A -85,B 0,C 180,E1 -27891.169,E2 -27891.169} C_VEL
LIN {X 0,Y 103.939,Z 360.021,A -85,B 0,C 180,E1 -27894.179,E2 -27894.179} C_VEL
LIN {X 0,Y 103.474,Z 359.478,A -85,B 0,C 180,E1 -27900.775,E2 -27900.775} C_VEL
LIN {X 0,Y 104.008,Z 360.15,A -85,B 0,C 180,E1 -27906.304,E2 -27906.304} C_VEL
LIN {X 0,Y 105.458,Z 363.703,A -85,B 0,C 180,E1 -27912.553,E2 -27912.553} C_VEL
LIN {X 0,Y 106.883,Z 365.167,A -85,B 0,C 180,E1 -27915.976,E2 -27915.976} C_VEL
LIN {X 0,Y 107.11,Z 365.732,A -85,B 0,C 180,E1 -27916.526,E2 -27916.526} C_VEL
LIN {X 0,Y 108.258,Z 368.929,A -85,B 0,C 180,E1 -27919.112,E2 -27919.112} C_VEL
LIN {X 0,Y 110.077,Z 375.667,A -85,B 0,C 180,E1 -27922.82,E2 -27922.82} C_VEL
LIN {X 0,Y 111.678,Z 381.487,A -85,B 0,C 180,E1 -27925.566,E2 -27925.566} C_VEL
LIN {X 0,Y 113.761,Z 386.881,A -85,B 0,C 180,E1 -27928.39,E2 -27928.39} C_VEL
LIN {X 0,Y 116.782,Z 393.495,A -85,B 0,C 180,E1 -27931.789,E2 -27931.789} C_VEL
LIN {X 0,Y 115.108,Z 406.313,A -85,B 0,C 180,E1 -27932.584,E2 -27932.584} C_VEL
LIN {X 0,Y 112.805,Z 416.223,A -85,B 0,C 180,E1 -27933.523,E2 -27933.523} C_VEL
LIN {X 0,Y 110.067,Z 424.972,A -85,B 0,C 180,E1 -27934.707,E2 -27934.707} C_VEL
LIN {X 0,Y 106.629,Z 433.688,A -85,B 0,C 180,E1 -27936.32,E2 -27936.32} C_VEL
LIN {X 0,Y 102.469,Z 442.316,A -85,B 0,C 180,E1 -27938.469,E2 -27938.469} C_VEL
LIN {X 0,Y 96.604,Z 452.141,A -85,B 0,C 180,E1 -27941.783,E2 -27941.783} C_VEL
LIN {X 0,Y 91.957,Z 458.777,A -85,B 0,C 180,E1 -27945.014,E2 -27945.014} C_VEL
LIN {X 0,Y 86.469,Z 465.471,A -85,B 0,C 180,E1 -27949.443,E2 -27949.443} C_VEL
LIN {X 0,Y 82.521,Z 469.877,A -85,B 0,C 180,E1 -27953.405,E2 -27953.405} C_VEL
LIN {X 0,Y 77.521,Z 475.063,A -85,B 0,C 180,E1 -27960.092,E2 -27960.092} C_VEL
LIN {X 0,Y 74.791,Z 477.72,A -85,B 0,C 180,E1 -27964.985,E2 -27964.985} C_VEL
LIN {X 0,Y 71.736,Z 480.633,A -85,B 0,C 180,E1 -27972.908,E2 -27972.908} C_VEL
LIN {X 0,Y 70.423,Z 481.9,A -85,B 0,C 180,E1 -27978.487,E2 -27978.487} C_VEL
LIN {X 0,Y 69.759,Z 482.696,A -85,B 0,C 180,E1 -27984.218,E2 -27984.218} C_VEL
LIN {X 0,Y 69.593,Z 482.999,A -85,B 0,C 180,E1 -27990,E2 -27990} C_VEL
LIN {X 0,Y 69.759,Z 482.715,A -85,B 0,C 180,E1 -27995.782,E2 -27995.782} C_VEL
LIN {X 0,Y 70.423,Z 481.956,A -85,B 0,C 180,E1 -28001.513,E2 -28001.513} C_VEL
LIN {X 0,Y 71.732,Z 480.726,A -85,B 0,C 180,E1 -28007.093,E2 -28007.093} C_VEL
LIN {X 0,Y 74.757,Z 477.853,A -85,B 0,C 180,E1 -28015.027,E2 -28015.027} C_VEL
LIN {X 0,Y 77.491,Z 475.236,A -85,B 0,C 180,E1 -28019.921,E2 -28019.921} C_VEL
LIN {X 0,Y 82.491,Z 470.098,A -85,B 0,C 180,E1 -28026.61,E2 -28026.61} C_VEL
LIN {X 0,Y 87.461,Z 464.571,A -85,B 0,C 180,E1 -28031.523,E2 -28031.523} C_VEL
LIN {X 0,Y 93.03,Z 457.62,A -85,B 0,C 180,E1 -28035.862,E2 -28035.862} C_VEL
LIN {X 0,Y 98.405,Z 449.643,A -85,B 0,C 180,E1 -28039.36,E2 -28039.36} C_VEL
LIN {X 0,Y 102.8,Z 442.107,A -85,B 0,C 180,E1 -28041.786,E2 -28041.786} C_VEL
LIN {X 0,Y 106.709,Z 434.063,A -85,B 0,C 180,E1 -28043.783,E2 -28043.783} C_VEL
LIN {X 0,Y 110.012,Z 425.814,A -85,B 0,C 180,E1 -28045.334,E2 -28045.334} C_VEL
LIN {X 0,Y 112.976,Z 416.352,A -85,B 0,C 180,E1 -28046.667,E2 -28046.667} C_VEL
LIN {X 0,Y 115.692,Z 404.701,A -85,B 0,C 180,E1 -28047.715,E2 -28047.715} C_VEL
LIN {X 0,Y 117.031,Z 393.748,A -85,B 0,C 180,E1 -28048.354,E2 -28048.354} C_VEL
LIN {X 0,Y 114.147,Z 387.367,A -85,B 0,C 180,E1 -28051.601,E2 -28051.601} C_VEL
LIN {X 0,Y 110.838,Z 381.041,A -85,B 0,C 180,E1 -28055.908,E2 -28055.908} C_VEL
LIN {X 0,Y 108.748,Z 377.422,A -85,B 0,C 180,E1 -28059.148,E2 -28059.148} C_VEL
LIN {X 0,Y 107.593,Z 375.413,A -85,B 0,C 180,E1 -28061.227,E2 -28061.227} C_VEL
LIN {X 0,Y 105.452,Z 371.653,A -85,B 0,C 180,E1 -28066.019,E2 -28066.019} C_VEL
LIN {X 0,Y 103.617,Z 368.92,A -85,B 0,C 180,E1 -28072.203,E2 -28072.203} C_VEL
LIN {X 0,Y 103.186,Z 367.079,A -85,B 0,C 180,E1 -28075.605,E2 -28075.605} C_VEL
LIN {X 0,Y 102.939,Z 366.592,A -85,B 0,C 180,E1 -28080,E2 -28080} C_VEL
LIN {X 0,Y 103.234,Z 367.336,A -85,B 0,C 180,E1 -28084.979,E2 -28084.979} C_VEL
LIN {X 0,Y 104.722,Z 370.972,A -85,B 0,C 180,E1 -28092.106,E2 -28092.106} C_VEL
LIN {X 0,Y 105.657,Z 372.034,A -85,B 0,C 180,E1 -28094.567,E2 -28094.567} C_VEL
LIN {X 0,Y 108.265,Z 376.531,A -85,B 0,C 180,E1 -28100.049,E2 -28100.049} C_VEL
LIN {X 0,Y 110.445,Z 380.296,A -85,B 0,C 180,E1 -28103.559,E2 -28103.559} C_VEL
LIN {X 0,Y 113.473,Z 386.024,A -85,B 0,C 180,E1 -28107.63,E2 -28107.63} C_VEL
LIN {X 0,Y 116.632,Z 392.792,A -85,B 0,C 180,E1 -28111.261,E2 -28111.261} C_VEL
LIN {X 0,Y 117.055,Z 393.782,A -85,B 0,C 180,E1 -28111.714,E2 -28111.714} C_VEL
LIN {X 0,Y 115.341,Z 406.495,A -85,B 0,C 180,E1 -28112.488,E2 -28112.488} C_VEL
LIN {X 0,Y 113.019,Z 416.331,A -85,B 0,C 180,E1 -28113.404,E2 -28113.404} C_VEL
LIN {X 0,Y 110.038,Z 425.709,A -85,B 0,C 180,E1 -28114.685,E2 -28114.685} C_VEL
LIN {X 0,Y 106.706,Z 433.978,A -85,B 0,C 180,E1 -28116.215,E2 -28116.215} C_VEL
LIN {X 0,Y 102.789,Z 442.05,A -85,B 0,C 180,E1 -28118.214,E2 -28118.214} C_VEL
LIN {X 0,Y 97.798,Z 450.605,A -85,B 0,C 180,E1 -28121.015,E2 -28121.015} C_VEL
LIN {X 0,Y 91.912,Z 459.058,A -85,B 0,C 180,E1 -28124.986,E2 -28124.986} C_VEL
LIN {X 0,Y 87.49,Z 464.536,A -85,B 0,C 180,E1 -28128.494,E2 -28128.494} C_VEL
LIN {X 0,Y 82.503,Z 470.069,A -85,B 0,C 180,E1 -28133.396,E2 -28133.396} C_VEL
LIN {X 0,Y 77.499,Z 475.213,A -85,B 0,C 180,E1 -28140.082,E2 -28140.082} C_VEL
LIN {X 0,Y 73.611,Z 478.986,A -85,B 0,C 180,E1 -28147.549,E2 -28147.549} C_VEL
LIN {X 0,Y 71.745,Z 480.714,A -85,B 0,C 180,E1 -28152.91,E2 -28152.91} C_VEL
LIN {X 0,Y 70.428,Z 481.948,A -85,B 0,C 180,E1 -28158.488,E2 -28158.488} C_VEL
LIN {X 0,Y 69.759,Z 482.712,A -85,B 0,C 180,E1 -28164.218,E2 -28164.218} C_VEL
LIN {X 0,Y 69.592,Z 483,A -85,B 0,C 180,E1 -28170,E2 -28170} C_VEL
LIN {X 0,Y 69.757,Z 482.699,A -85,B 0,C 180,E1 -28175.782,E2 -28175.782} C_VEL
LIN {X 0,Y 70.421,Z 481.907,A -85,B 0,C 180,E1 -28181.513,E2 -28181.513} C_VEL
LIN {X 0,Y 71.731,Z 480.645,A -85,B 0,C 180,E1 -28187.093,E2 -28187.093} C_VEL
LIN {X 0,Y 74.766,Z 477.738,A -85,B 0,C 180,E1 -28195.023,E2 -28195.023} C_VEL
LIN {X 0,Y 77.493,Z 475.086,A -85,B 0,C 180,E1 -28199.92,E2 -28199.92} C_VEL
LIN {X 0,Y 82.5,Z 469.906,A -85,B 0,C 180,E1 -28206.605,E2 -28206.605} C_VEL
LIN {X 0,Y 88.56,Z 463.067,A -85,B 0,C 180,E1 -28212.418,E2 -28212.418} C_VEL
LIN {X 0,Y 94.181,Z 455.597,A -85,B 0,C 180,E1 -28216.681,E2 -28216.681} C_VEL
LIN {X 0,Y 99.041,Z 448.226,A -85,B 0,C 180,E1 -28219.713,E2 -28219.713} C_VEL
LIN {X 0,Y 103.359,Z 440.546,A -85,B 0,C 180,E1 -28222.085,E2 -28222.085} C_VEL
LIN {X 0,Y 107.338,Z 431.97,A -85,B 0,C 180,E1 -28224.119,E2 -28224.119} C_VEL
LIN {X 0,Y 111.19,Z 421.728,A -85,B 0,C 180,E1 -28225.872,E2 -28225.872} C_VEL
LIN {X 0,Y 114.289,Z 410.241,A -85,B 0,C 180,E1 -28227.14,E2 -28227.14} C_VEL
LIN {X 0,Y 116.064,Z 400.517,A -85,B 0,C 180,E1 -28227.815,E2 -28227.815} C_VEL
LIN {X 0,Y 116.827,Z 393.54,A -85,B 0,C 180,E1 -28228.215,E2 -28228.215} C_VEL
LIN {X 0,Y 113.331,Z 386.024,A -85,B 0,C 180,E1 -28232.174,E2 -28232.174} C_VEL
LIN {X 0,Y 110.574,Z 380.762,A -85,B 0,C 180,E1 -28235.816,E2 -28235.816} C_VEL
LIN {X 0,Y 108.499,Z 377.184,A -85,B 0,C 180,E1 -28239.021,E2 -28239.021} C_VEL
LIN {X 0,Y 107.195,Z 375.003,A -85,B 0,C 180,E1 -28241.361,E2 -28241.361} C_VEL
LIN {X 0,Y 105.266,Z 371.555,A -85,B 0,C 180,E1 -28245.674,E2 -28245.674} C_VEL
LIN {X 0,Y 103.419,Z 368.865,A -85,B 0,C 180,E1 -28251.636,E2 -28251.636} C_VEL
LIN {X 0,Y 102.928,Z 366.945,A -85,B 0,C 180,E1 -28255.104,E2 -28255.104} C_VEL
LIN {X 0,Y 102.61,Z 366.448,A -85,B 0,C 180,E1 -28260,E2 -28260} C_VEL
LIN {X 0,Y 103.015,Z 367.159,A -85,B 0,C 180,E1 -28265.629,E2 -28265.629} C_VEL
LIN {X 0,Y 104.338,Z 370.617,A -85,B 0,C 180,E1 -28271.916,E2 -28271.916} C_VEL
LIN {X 0,Y 105.491,Z 372.002,A -85,B 0,C 180,E1 -28274.958,E2 -28274.958} C_VEL
LIN {X 0,Y 108.101,Z 376.445,A -85,B 0,C 180,E1 -28280.33,E2 -28280.33} C_VEL
LIN {X 0,Y 110.264,Z 380.192,A -85,B 0,C 180,E1 -28283.778,E2 -28283.778} C_VEL
LIN {X 0,Y 113.212,Z 385.772,A -85,B 0,C 180,E1 -28287.723,E2 -28287.723} C_VEL
LIN {X 0,Y 113.761,Z 386.881,A -85,B 0,C 180,E1 -28288.39,E2 -28288.39} C_VEL
LIN {X 0,Y 114.431,Z 389.39,A -85,B 0,C 180,E1 -28289.31,E2 -28289.31} C_VEL
LIN {X 0,Y 114.53,Z 393.15,A -85,B 0,C 180,E1 -28289.859,E2 -28289.859} C_VEL
LIN {X 0,Y 113.824,Z 397.894,A -85,B 0,C 180,E1 -28289.925,E2 -28289.925} C_VEL
LIN {X 0,Y 111.492,Z 406.447,A -85,B 0,C 180,E1 -28289.571,E2 -28289.571} C_VEL
LIN {X 0,Y 111.11,Z 407.875,A -85,B 0,C 180,E1 -28289.629,E2 -28289.629} C_VEL
LIN {X 0,Y 109.191,Z 415.756,A -85,B 0,C 180,E1 -28290.364,E2 -28290.364} C_VEL
LIN {X 0,Y 106.195,Z 424.976,A -85,B 0,C 180,E1 -28291.565,E2 -28291.565} C_VEL
LIN {X 0,Y 102.728,Z 433.39,A -85,B 0,C 180,E1 -28293.065,E2 -28293.065} C_VEL
LIN {X 0,Y 98.761,Z 441.324,A -85,B 0,C 180,E1 -28294.961,E2 -28294.961} C_VEL
LIN {X 0,Y 93.966,Z 449.191,A -85,B 0,C 180,E1 -28297.377,E2 -28297.377} C_VEL
LIN {X 0,Y 88.321,Z 457.25,A -85,B 0,C 180,E1 -28300.893,E2 -28300.893} C_VEL
LIN {X 0,Y 82.342,Z 464.301,A -85,B 0,C 180,E1 -28305.241,E2 -28305.241} C_VEL
LIN {X 0,Y 76.936,Z 469.879,A -85,B 0,C 180,E1 -28310.251,E2 -28310.251} C_VEL
LIN {X 0,Y 71.454,Z 475.064,A -85,B 0,C 180,E1 -28317.252,E2 -28317.252} C_VEL
LIN {X 0,Y 68.428,Z 477.721,A -85,B 0,C 180,E1 -28322.473,E2 -28322.473} C_VEL
LIN {X 0,Y 64.991,Z 480.633,A -85,B 0,C 180,E1 -28331.07,E2 -28331.07} C_VEL
LIN {X 0,Y 63.485,Z 481.9,A -85,B 0,C 180,E1 -28337.209,E2 -28337.209} C_VEL
LIN {X 0,Y 62.689,Z 482.696,A -85,B 0,C 180,E1 -28343.563,E2 -28343.563} C_VEL
LIN {X 0,Y 62.512,Z 482.999,A -85,B 0,C 180,E1 -28350,E2 -28350} C_VEL
LIN {X 0,Y 62.689,Z 482.715,A -85,B 0,C 180,E1 -28356.437,E2 -28356.437} C_VEL
LIN {X 0,Y 63.484,Z 481.955,A -85,B 0,C 180,E1 -28362.792,E2 -28362.792} C_VEL
LIN {X 0,Y 64.986,Z 480.725,A -85,B 0,C 180,E1 -28368.931,E2 -28368.931} C_VEL
LIN {X 0,Y 68.378,Z 477.852,A -85,B 0,C 180,E1 -28377.549,E2 -28377.549} C_VEL
LIN {X 0,Y 71.405,Z 475.235,A -85,B 0,C 180,E1 -28382.774,E2 -28382.774} C_VEL
LIN {X 0,Y 76.905,Z 470.096,A -85,B 0,C 180,E1 -28389.768,E2 -28389.768} C_VEL
LIN {X 0,Y 82.279,Z 464.569,A -85,B 0,C 180,E1 -28394.803,E2 -28394.803} C_VEL
LIN {X 0,Y 88.229,Z 457.618,A -85,B 0,C 180,E1 -28399.176,E2 -28399.176} C_VEL
LIN {X 0,Y 93.948,Z 449.64,A -85,B 0,C 180,E1 -28402.637,E2 -28402.637} C_VEL
LIN {X 0,Y 98.747,Z 441.79,A -85,B 0,C 180,E1 -28405.107,E2 -28405.107} C_VEL
LIN {X 0,Y 102.681,Z 434.058,A -85,B 0,C 180,E1 -28406.975,E2 -28406.975} C_VEL
LIN {X 0,Y 106.132,Z 425.808,A -85,B 0,C 180,E1 -28408.491,E2 -28408.491} C_VEL
LIN {X 0,Y 108.906,Z 417.511,A -85,B 0,C 180,E1 -28409.635,E2 -28409.635} C_VEL
LIN {X 0,Y 111.222,Z 408.534,A -85,B 0,C 180,E1 -28410.494,E2 -28410.494} C_VEL
LIN {X 0,Y 112.868,Z 399.099,A -85,B 0,C 180,E1 -28411.102,E2 -28411.102} C_VEL
LIN {X 0,Y 113.102,Z 396.572,A -85,B 0,C 180,E1 -28411.336,E2 -28411.336} C_VEL
LIN {X 0,Y 109.977,Z 389.64,A -85,B 0,C 180,E1 -28415.566,E2 -28415.566} C_VEL
LIN {X 0,Y 107.433,Z 384.652,A -85,B 0,C 180,E1 -28419.663,E2 -28419.663} C_VEL
LIN {X 0,Y 105.887,Z 381.806,A -85,B 0,C 180,E1 -28422.676,E2 -28422.676} C_VEL
LIN {X 0,Y 104.045,Z 378.336,A -85,B 0,C 180,E1 -28427.318,E2 -28427.318} C_VEL
LIN {X 0,Y 102.395,Z 375.125,A -85,B 0,C 180,E1 -28434.337,E2 -28434.337} C_VEL
LIN {X 0,Y 102.259,Z 374.128,A -85,B 0,C 180,E1 -28436.059,E2 -28436.059} C_VEL
LIN {X 0,Y 102.074,Z 373.64,A -85,B 0,C 180,E1 -28440,E2 -28440} C_VEL
LIN {X 0,Y 102.269,Z 374.277,A -85,B 0,C 180,E1 -28444.211,E2 -28444.211} C_VEL
LIN {X 0,Y 103.698,Z 377.986,A -85,B 0,C 180,E1 -28451.731,E2 -28451.731} C_VEL
LIN {X 0,Y 104.357,Z 378.91,A -85,B 0,C 180,E1 -28453.633,E2 -28453.633} C_VEL
LIN {X 0,Y 106.567,Z 383.016,A -85,B 0,C 180,E1 -28458.753,E2 -28458.753} C_VEL
LIN {X 0,Y 108.661,Z 386.977,A -85,B 0,C 180,E1 -28462.458,E2 -28462.458} C_VEL
LIN {X 0,Y 111.497,Z 392.833,A -85,B 0,C 180,E1 -28466.598,E2 -28466.598} C_VEL
LIN {X 0,Y 113.153,Z 396.742,A -85,B 0,C 180,E1 -28468.786,E2 -28468.786} C_VEL
LIN {X 0,Y 111.693,Z 406.515,A -85,B 0,C 180,E1 -28469.422,E2 -28469.422} C_VEL
LIN {X 0,Y 109.414,Z 415.856,A -85,B 0,C 180,E1 -28470.241,E2 -28470.241} C_VEL
LIN {X 0,Y 106.853,Z 423.842,A -85,B 0,C 180,E1 -28471.238,E2 -28471.238} C_VEL
LIN {X 0,Y 103.376,Z 432.483,A -85,B 0,C 180,E1 -28472.723,E2 -28472.723} C_VEL
LIN {X 0,Y 99.267,Z 440.778,A -85,B 0,C 180,E1 -28474.636,E2 -28474.636} C_VEL
LIN {X 0,Y 94.627,Z 448.568,A -85,B 0,C 180,E1 -28477.023,E2 -28477.023} C_VEL
LIN {X 0,Y 89.457,Z 455.885,A -85,B 0,C 180,E1 -28480.007,E2 -28480.007} C_VEL
LIN {X 0,Y 83.458,Z 463.305,A -85,B 0,C 180,E1 -28484.294,E2 -28484.294} C_VEL
LIN {X 0,Y 77.949,Z 469.116,A -85,B 0,C 180,E1 -28489.182,E2 -28489.182} C_VEL
LIN {X 0,Y 73.096,Z 473.698,A -85,B 0,C 180,E1 -28494.769,E2 -28494.769} C_VEL
